// TIA Portal project "Szachy_v2" (V14)

(* hardware
DEVICE "S71500/ET200MP station_1"  S7-1500 station
   slot 0: "Rail_0"  Rack  6ES7 590-1***0-0AA0
   slot 1: "PLC_1"  CPU 1511-1 PN  6ES7 511-1AK00-0AB0  V1.8
      slot 3: "CPU display_1"  6ES7591-1AA00-0AA0
   slot 2: "DI 16x24VDC HF_1"  DI 16x24VDC HF  6ES7 521-1BH00-0AB0  V2.1
   slot 3: "DQ 16x24VDC/0.5A ST_1"  DQ 16x24VDC/0.5A ST  6ES7 522-1BH00-0AB0  V2.0
   slot 4: "AI 4xU/I/RTD/TC ST_1"  AI 4xU/I/RTD/TC ST  6ES7 531-7QD00-0AB0  V1.0
DEVICE "HMI_1"  TP700 Comfort
   slot 0: "TP700 Comfort"  TP700 Comfort  6AV2 124-0GC01-0AX0  14.0.1.0
   slot 1: "HMI_RT_1"  TP700 Comfort  6AV2 124-0GC01-0AX0  14.0.1.0
   slot 5: "HMI_1.IE_CP_1"  PROFINET Interface  14.0.1.0
      slot 1: "PROFINET Interface_1"  PROFINET Interface
         slot 1: "Port_1"  Port
         slot 2: "Port_2"  Port
   slot 7: "HMI_1.MPI/DP_CP_1"  MPI/DP Interface  14.0.1.0
*)

// ===== PLC "PLC_1"  CPU 1511-1 PN =====

VAR_GLOBAL   // PLC tag table "Default tag table"
   "Tag_1" AT %M100.0 : Bool;
   "Tag_2" AT %M100.1 : Bool;
END_VAR

TYPE "Szachownica"
   STRUCT
      figury : Array[0..31] of "Figura";
      pozycja_wybranego_1 : "Pozycja";
      pozycja_wybranego_2 : "Pozycja";
   END_STRUCT;
END_TYPE

TYPE "Figura"
   STRUCT
      kolor : Bool;   // 0-czarny / 1-biały
      rodzaj : Int;   // 0-pawn /1-bishop /2-horse /3-tower / 4-queen /5-king
      zywy : Bool;   // 1-zywy /0-zbity
      mozliwe_ruchy : Array[0..26] of "Pozycja";
      pozycja : "Pozycja";
      poczatkowa_pozycja : Bool := true;
      tura_1_ruchu_piona : Int;
   END_STRUCT;
END_TYPE

TYPE "Pozycja"
   STRUCT
      x : Int;
      y : Int;
   END_STRUCT;
END_TYPE

DATA_BLOCK "StatusyHMI"   // DB1
{ S7_Optimized_Access := 'FALSE' }
VERSION : 0.1
   VAR
      przyciski : Array[0..63] of Bool;
      "statusy figur" : Array[0..63] of Int;
      "przyciski widocznosc" : Array[0..63] of Bool;
   END_VAR
BEGIN
   "przyciski widocznosc"[0] := true;
   "przyciski widocznosc"[1] := true;
   "przyciski widocznosc"[2] := true;
   "przyciski widocznosc"[3] := true;
   "przyciski widocznosc"[4] := true;
   "przyciski widocznosc"[5] := true;
   "przyciski widocznosc"[6] := true;
   "przyciski widocznosc"[7] := true;
   "przyciski widocznosc"[8] := true;
   "przyciski widocznosc"[9] := true;
   "przyciski widocznosc"[10] := true;
   "przyciski widocznosc"[11] := true;
   "przyciski widocznosc"[12] := true;
   "przyciski widocznosc"[13] := true;
   "przyciski widocznosc"[14] := true;
   "przyciski widocznosc"[15] := true;
   "przyciski widocznosc"[16] := true;
   "przyciski widocznosc"[17] := true;
   "przyciski widocznosc"[18] := true;
   "przyciski widocznosc"[19] := true;
   "przyciski widocznosc"[20] := true;
   "przyciski widocznosc"[21] := true;
   "przyciski widocznosc"[22] := true;
   "przyciski widocznosc"[23] := true;
   "przyciski widocznosc"[24] := true;
   "przyciski widocznosc"[25] := true;
   "przyciski widocznosc"[26] := true;
   "przyciski widocznosc"[27] := true;
   "przyciski widocznosc"[28] := true;
   "przyciski widocznosc"[29] := true;
   "przyciski widocznosc"[30] := true;
   "przyciski widocznosc"[31] := true;
   "przyciski widocznosc"[32] := true;
   "przyciski widocznosc"[33] := true;
   "przyciski widocznosc"[34] := true;
   "przyciski widocznosc"[35] := true;
   "przyciski widocznosc"[36] := true;
   "przyciski widocznosc"[37] := true;
   "przyciski widocznosc"[38] := true;
   "przyciski widocznosc"[39] := true;
   "przyciski widocznosc"[40] := true;
   "przyciski widocznosc"[41] := true;
   "przyciski widocznosc"[42] := true;
   "przyciski widocznosc"[43] := true;
   "przyciski widocznosc"[44] := true;
   "przyciski widocznosc"[45] := true;
   "przyciski widocznosc"[46] := true;
   "przyciski widocznosc"[47] := true;
   "przyciski widocznosc"[48] := true;
   "przyciski widocznosc"[49] := true;
   "przyciski widocznosc"[50] := true;
   "przyciski widocznosc"[51] := true;
   "przyciski widocznosc"[52] := true;
   "przyciski widocznosc"[53] := true;
   "przyciski widocznosc"[54] := true;
   "przyciski widocznosc"[55] := true;
   "przyciski widocznosc"[56] := true;
   "przyciski widocznosc"[57] := true;
   "przyciski widocznosc"[58] := true;
   "przyciski widocznosc"[59] := true;
   "przyciski widocznosc"[60] := true;
   "przyciski widocznosc"[61] := true;
   "przyciski widocznosc"[62] := true;
   "przyciski widocznosc"[63] := true;
   "statusy figur"[0] := 12;
   "statusy figur"[1] := 12;
   "statusy figur"[2] := 12;
   "statusy figur"[3] := 12;
   "statusy figur"[4] := 12;
   "statusy figur"[5] := 12;
   "statusy figur"[6] := 12;
   "statusy figur"[7] := 12;
   "statusy figur"[8] := 12;
   "statusy figur"[9] := 12;
   "statusy figur"[10] := 12;
   "statusy figur"[11] := 12;
   "statusy figur"[12] := 12;
   "statusy figur"[13] := 12;
   "statusy figur"[14] := 12;
   "statusy figur"[15] := 12;
   "statusy figur"[16] := 12;
   "statusy figur"[17] := 12;
   "statusy figur"[18] := 12;
   "statusy figur"[19] := 12;
   "statusy figur"[20] := 12;
   "statusy figur"[21] := 12;
   "statusy figur"[22] := 12;
   "statusy figur"[23] := 12;
   "statusy figur"[24] := 12;
   "statusy figur"[25] := 12;
   "statusy figur"[26] := 12;
   "statusy figur"[27] := 12;
   "statusy figur"[28] := 12;
   "statusy figur"[29] := 12;
   "statusy figur"[30] := 12;
   "statusy figur"[31] := 12;
   "statusy figur"[32] := 12;
   "statusy figur"[33] := 12;
   "statusy figur"[34] := 12;
   "statusy figur"[35] := 12;
   "statusy figur"[36] := 12;
   "statusy figur"[37] := 12;
   "statusy figur"[38] := 12;
   "statusy figur"[39] := 12;
   "statusy figur"[40] := 12;
   "statusy figur"[41] := 12;
   "statusy figur"[42] := 12;
   "statusy figur"[43] := 12;
   "statusy figur"[44] := 12;
   "statusy figur"[45] := 12;
   "statusy figur"[46] := 12;
   "statusy figur"[47] := 12;
   "statusy figur"[48] := 12;
   "statusy figur"[49] := 12;
   "statusy figur"[50] := 12;
   "statusy figur"[51] := 12;
   "statusy figur"[52] := 12;
   "statusy figur"[53] := 12;
   "statusy figur"[54] := 12;
   "statusy figur"[55] := 12;
   "statusy figur"[56] := 12;
   "statusy figur"[57] := 12;
   "statusy figur"[58] := 12;
   "statusy figur"[59] := 12;
   "statusy figur"[60] := 12;
   "statusy figur"[61] := 12;
   "statusy figur"[62] := 12;
   "statusy figur"[63] := 12;
END_DATA_BLOCK

DATA_BLOCK "Historia_gry"   // DB3
{ S7_Optimized_Access := 'TRUE' }
VERSION : 0.1
   VAR
      stan_figur : Array[0..200] of "Szachownica";
      indeks_historii : Int := 0;
   END_VAR
BEGIN
END_DATA_BLOCK

DATA_BLOCK "Status_rozgrywki"   // DB4
{ S7_Optimized_Access := 'TRUE' }
VERSION : 0.1
   VAR
      tura_int : Int;
      inicjalizacja : Bool := true;
      Szachownica : "Szachownica";
      tura_bool : Bool := true;   // true - biale false -czarne
      szach_biale : Bool;
      szach_czarne : Bool;
      szachmat_biale : Bool;
      szachmat_czarne : Bool;
      remis : Bool;   // 1- remis, 0 - nie stwierdzono
      status_zakonczenia_gry : Bool;   // 0 - trwa, 1-zakonczono
      komunikat_koniec_gry : Int;   // 0 - wygrana białe, 1- czarne , 2 -remis
      wybrano_pierwszy : Bool;
      indeks1 : Int := -1;
      indeks2 : Int := -2;
      wybrano_drugi : Bool;
   END_VAR
BEGIN
END_DATA_BLOCK

DATA_BLOCK "Inicjalizacja_DB"   // DB5
{ S7_Optimized_Access := 'TRUE' }
VERSION : 0.1
// stored: InstanceOfName Inicjalizacja
"Inicjalizacja"
BEGIN
   Fig_init.figury[7].pozycja.y := 1;
   Fig_init.figury[7].pozycja.x := 8;
   Fig_init.figury[12].pozycja.y := 2;
END_DATA_BLOCK

DATA_BLOCK "sprawdz_czy_remis_DB"   // DB7
{ S7_Optimized_Access := 'TRUE' }
VERSION : 0.1
// stored: InstanceOfName sprawdz_czy_remis
"sprawdz_czy_remis"
BEGIN
END_DATA_BLOCK

// folder: AI

DATA_BLOCK "Ruchy_AI"   // DB8
{ S7_Optimized_Access := 'TRUE' }
VERSION : 0.1
   VAR
      ruchy_1 : Array[0..1] of Bool;
   END_VAR
BEGIN
END_DATA_BLOCK

// folder: (top level)

FUNCTION_BLOCK "Inicjalizacja"   // FB1, SCL
{ S7_Optimized_Access := 'TRUE' }
VERSION : 0.1
   VAR RETAIN
      Fig_init : "Szachownica";
   END_VAR
   VAR
      biale_init : Bool;
   END_VAR
   // Fig_init.figury[0].kolor := 1;
   // Fig_init.figury[0].rodzaj := 3;
   // Fig_init.figury[0].zywy := 1;
   // Fig_init.figury[1].rodzaj := 2;
   // Fig_init.figury[2].rodzaj := 1;
   // Fig_init.figury[3].rodzaj := 4;
   // Fig_init.figury[4].rodzaj := 5;
   // Fig_init.figury[5].rodzaj := 1;
   // Fig_init.figury[6].rodzaj := 2;
   // Fig_init.figury[7].rodzaj := 3;
   // Fig_init.figury[1].zywy := 1;
   // Fig_init.figury[2].zywy := 1;
   // Fig_init.figury[3].zywy := 1;
   // Fig_init.figury[4].zywy := 1;
   // Fig_init.figury[5].zywy := 1;
   // Fig_init.figury[6].zywy := 1;
   // Fig_init.figury[7].zywy := 1;
   // Fig_init.figury[7].kolor := 1;
   // Fig_init.figury[6].kolor := 1;
   // Fig_init.figury[5].kolor := 1;
   // Fig_init.figury[4].kolor := 1;
   // Fig_init.figury[3].kolor := 1;
   // Fig_init.figury[2].kolor := 1;
   // Fig_init.figury[1].kolor := 1;
   // Fig_init.figury[1].pozycja.x := 2;
   // Fig_init.figury[2].pozycja.x := 3;
   // Fig_init.figury[3].pozycja.x := 4;
   // Fig_init.figury[4].pozycja.x := 5;
   // Fig_init.figury[5].pozycja.x := 6;
   // Fig_init.figury[6].pozycja.x := 7;
   // Fig_init.figury[7].pozycja.x := 7;
   // Fig_init.figury[8].pozycja.x := 1;
   // Fig_init.figury[0].pozycja.x := 1;
   // Fig_init.figury[0].pozycja.y := 1;
   // Fig_init.figury[1].pozycja.y := 1;
   // Fig_init.figury[2].pozycja.y := 1;
   // Fig_init.figury[3].pozycja.y := 1;
   // Fig_init.figury[4].pozycja.y := 1;
   // Fig_init.figury[5].pozycja.y := 1;
   // Fig_init.figury[6].pozycja.y := 1;
   // Fig_init.figury[8].kolor := 1;
   // Fig_init.figury[8].zywy := 1;
   // Fig_init.figury[8].pozycja.y := 2;
   // Fig_init.figury[9].kolor := 1;
   // Fig_init.figury[9].rodzaj := 0;
   // Fig_init.figury[9].zywy := 1;
   // Fig_init.figury[10].kolor := 1;
   // Fig_init.figury[10].rodzaj := 0;
   // Fig_init.figury[10].zywy := 1;
   // Fig_init.figury[11].kolor := 1;
   // Fig_init.figury[11].rodzaj := 0;
   // Fig_init.figury[11].zywy := 1;
   // Fig_init.figury[12].kolor := 1;
   // Fig_init.figury[12].rodzaj := 0;
   // Fig_init.figury[12].zywy := 1;
   // Fig_init.figury[13].kolor := 1;
   // Fig_init.figury[13].rodzaj := 0;
   // Fig_init.figury[13].zywy := 1;
   // Fig_init.figury[14].kolor := 1;
   // Fig_init.figury[14].rodzaj := 0;
   // Fig_init.figury[14].zywy := 1;
   // Fig_init.figury[15].kolor := 1;
   // Fig_init.figury[15].rodzaj := 0;
   // Fig_init.figury[15].zywy := 1;
   // Fig_init.figury[9].pozycja.x := 2;
   // Fig_init.figury[9].pozycja.y := 2;
   // Fig_init.figury[10].pozycja.x := 3;
   // Fig_init.figury[10].pozycja.y := 2;
   // Fig_init.figury[11].pozycja.x := 4;
   // Fig_init.figury[11].pozycja.y := 2;
   // Fig_init.figury[12].pozycja.x := 5;
   // Fig_init.figury[13].pozycja.x := 6;
   // Fig_init.figury[13].pozycja.y := 2;
   // Fig_init.figury[14].pozycja.x := 7;
   // Fig_init.figury[14].pozycja.y := 2;
   // Fig_init.figury[15].pozycja.x := 8;
   // Fig_init.figury[15].pozycja.y := 2;
   // Fig_init.figury[16].kolor := 0;
   // Fig_init.figury[16].zywy := 1;
   // Fig_init.figury[17].kolor := 0;
   // Fig_init.figury[17].rodzaj := 0;
   // Fig_init.figury[17].zywy := 1;
   // Fig_init.figury[23].kolor := 0;
   // Fig_init.figury[23].rodzaj := 0;
   // Fig_init.figury[23].zywy := 1;
   // Fig_init.figury[18].kolor := 0;
   // Fig_init.figury[18].rodzaj := 0;
   // Fig_init.figury[18].zywy := 1;
   // Fig_init.figury[19].kolor := 0;
   // Fig_init.figury[19].rodzaj := 0;
   // Fig_init.figury[19].zywy := 1;
   // Fig_init.figury[22].kolor := 0;
   // Fig_init.figury[22].rodzaj := 0;
   // Fig_init.figury[22].zywy := 1;
   // Fig_init.figury[21].kolor := 0;
   // Fig_init.figury[21].rodzaj := 0;
   // Fig_init.figury[21].zywy := 1;
   // Fig_init.figury[20].kolor := 0;
   // Fig_init.figury[20].rodzaj := 0;
   // Fig_init.figury[20].zywy := 1;
   // Fig_init.figury[16].pozycja.x := 1;
   // Fig_init.figury[16].pozycja.y := 7;
   // Fig_init.figury[17].pozycja.x := 2;
   // Fig_init.figury[17].pozycja.y := 7;
   // Fig_init.figury[18].pozycja.x := 3;
   // Fig_init.figury[18].pozycja.y := 7;
   // Fig_init.figury[19].pozycja.x := 4;
   // Fig_init.figury[19].pozycja.y := 7;
   // Fig_init.figury[20].pozycja.x := 5;
   // Fig_init.figury[20].pozycja.y := 7;
   // Fig_init.figury[21].pozycja.x := 6;
   // Fig_init.figury[21].pozycja.y := 7;
   // Fig_init.figury[22].pozycja.x := 7;
   // Fig_init.figury[22].pozycja.y := 7;
   // Fig_init.figury[23].pozycja.x := 8;
   // Fig_init.figury[23].pozycja.y := 7;
   // Fig_init.figury[24].kolor := 0;
   // Fig_init.figury[24].zywy := 1;
   // Fig_init.figury[24].rodzaj := 3;
   // Fig_init.figury[25].kolor := 0;
   // Fig_init.figury[25].rodzaj := 2;
   // Fig_init.figury[25].zywy := 1;
   // Fig_init.figury[24].pozycja.x := 1;
   // Fig_init.figury[24].pozycja.y := 8;
   // Fig_init.figury[25].pozycja.x := 2;
   // Fig_init.figury[25].pozycja.y := 8;
   // Fig_init.figury[26].kolor := 0;
   // Fig_init.figury[26].rodzaj := 1;
   // Fig_init.figury[26].zywy := 1;
   // Fig_init.figury[26].pozycja.x := 3;
   // Fig_init.figury[26].pozycja.y := 8;
   // Fig_init.figury[27].kolor := 0;
   // Fig_init.figury[27].rodzaj := 4;
   // Fig_init.figury[27].zywy := 1;
   // Fig_init.figury[27].pozycja.x := 4;
   // Fig_init.figury[27].pozycja.y := 8;
   // Fig_init.figury[28].kolor := 0;
   // Fig_init.figury[28].rodzaj := 5;
   // Fig_init.figury[28].zywy := 1;
   // Fig_init.figury[28].pozycja.x := 5;
   // Fig_init.figury[28].pozycja.y := 8;
   // Fig_init.figury[29].kolor := 0;
   // Fig_init.figury[29].rodzaj := 1;
   // Fig_init.figury[29].zywy := 1;
   // Fig_init.figury[29].pozycja.x := 6;
   // Fig_init.figury[29].pozycja.y := 8;
   // Fig_init.figury[30].kolor := 0;
   // Fig_init.figury[30].rodzaj := 2;
   // Fig_init.figury[30].zywy := 1;
   // Fig_init.figury[30].pozycja.x := 7;
   // Fig_init.figury[30].pozycja.y := 8;
   // Fig_init.figury[31].kolor := 0;
   // Fig_init.figury[31].rodzaj := 3;
   // Fig_init.figury[31].zywy := 1;
   // Fig_init.figury[31].pozycja.x := 8;
   // Fig_init.figury[31].pozycja.y := 8;
BEGIN
   "Historia_gry".stan_figur[0] := #Fig_init;
   "Status_rozgrywki".Szachownica := #Fig_init;
   "Status_rozgrywki".tura_int := 1;
   "Status_rozgrywki".inicjalizacja := false;
   "Status_rozgrywki".tura_bool := TRUE;
   "Czyszczenie_mozliwych_ruchów"();
   "Czyszczenie_podświetlenia"();
   #biale_init := TRUE;
   "Status_rozgrywki".szach_biale := 0;
   "Status_rozgrywki".szach_czarne := 0;
   "Status_rozgrywki".szachmat_biale := 0;
   "Status_rozgrywki".szachmat_czarne := 0;
   "Status_rozgrywki".status_zakonczenia_gry := 0;
   "Status_rozgrywki".komunikat_koniec_gry := 0;
END_FUNCTION_BLOCK

FUNCTION "tura_biale" : Void   // FC1, SCL
{ S7_Optimized_Access := 'TRUE' }
VERSION : 0.1
   VAR_IN_OUT
      tura : Bool;
   END_VAR
   VAR_TEMP
      ilosc_mozliwych_ruchow : Int;
      figura_ruch : "Figura";
      tura_zbocze : Bool;
   END_VAR
BEGIN
   "tura_biale_trig_DB"(CLK := #tura,
                         Q => #tura_zbocze);
   //"Status_rozgrywki".szach_biale := "sprawdz_czy_szach"(tura_bool := TRUE, szachownica := "Status_rozgrywki".Szachownica);
   //#ilosc_mozliwych_ruchow := "Wykrywanie_ruchów"(tura_bool := TRUE, Szachownica := "Status_rozgrywki".Szachownica);
   //"Status_rozgrywki".szachmat_biale := (#ilosc_mozliwych_ruchow = 0);

    IF #tura_zbocze OR "Inicjalizacja_DB".biale_init THEN
           "Status_rozgrywki".szach_biale := "sprawdz_czy_szach"(tura_bool := TRUE, szachownica := "Status_rozgrywki".Szachownica);
           #ilosc_mozliwych_ruchow := "Wykrywanie_ruchów"(tura_bool := TRUE, Szachownica := "Status_rozgrywki".Szachownica);
           "Status_rozgrywki".szachmat_biale := (#ilosc_mozliwych_ruchow = 0 AND "Status_rozgrywki".szach_biale);

           "Inicjalizacja_DB".biale_init := FALSE;
       END_IF;
    IF #tura THEN
       IF "Status_rozgrywki".wybrano_pierwszy AND "Status_rozgrywki".wybrano_drugi THEN
           IF "konwersja_pozycja_na_figura"(pozycja := "Status_rozgrywki".Szachownica.pozycja_wybranego_1,
                                                Szachownica := "Status_rozgrywki".Szachownica, figura => #figura_ruch) THEN
               IF "sprawdz_czy_ruch_mozliwy"(Szachownica := "Status_rozgrywki".Szachownica, figura := #figura_ruch, pozycja := "Status_rozgrywki".Szachownica.pozycja_wybranego_2) THEN
                   "wykonanie_ruchu"(pozycja := "Status_rozgrywki".Szachownica.pozycja_wybranego_2,
                                     szachownica := "Status_rozgrywki".Szachownica,
                                     figura := #figura_ruch);
                   "Czyszczenie_podświetlenia"();
                   "Czyszczenie_mozliwych_ruchów"();
                   "Status_rozgrywki".tura_int += 1;
                   "Status_rozgrywki".szach_biale := 0;
                   #tura := false;
               END_IF;
           END_IF;
       END_IF;
   END_IF;
END_FUNCTION

FUNCTION "tura_czarne" : Void   // FC2, SCL
{ S7_Optimized_Access := 'TRUE' }
VERSION : 0.1
   VAR_IN_OUT
      tura : Bool;
   END_VAR
   VAR_TEMP
      ilosc_mozliwych_ruchow : Int;
      figura_ruch : "Figura";
      tura_zbocze : Bool;
   END_VAR
BEGIN
   "Tura_czarne_trug_DB"(CLK:=#tura,
                         Q=>#tura_zbocze);
   //"Status_rozgrywki".szach_czarne := "sprawdz_czy_szach"(tura_bool := FALSE, szachownica := "Status_rozgrywki".Szachownica);
   //#ilosc_mozliwych_ruchow := "Wykrywanie_ruchów"(tura_bool := FALSE, Szachownica := "Status_rozgrywki".Szachownica);
   //"Status_rozgrywki".szachmat_czarne := (#ilosc_mozliwych_ruchow = 0);
   IF #tura_zbocze THEN
       "Status_rozgrywki".szach_czarne := "sprawdz_czy_szach"(tura_bool := FALSE, szachownica := "Status_rozgrywki".Szachownica);
       #ilosc_mozliwych_ruchow := "Wykrywanie_ruchów"(tura_bool := FALSE, Szachownica := "Status_rozgrywki".Szachownica);
       "Status_rozgrywki".szachmat_czarne := (#ilosc_mozliwych_ruchow = 0 AND "Status_rozgrywki".szach_czarne);
       "sprawdz_czy_remis_DB"(#ilosc_mozliwych_ruchow);
   END_IF;
   IF NOT #tura THEN
       IF "Status_rozgrywki".wybrano_pierwszy AND "Status_rozgrywki".wybrano_drugi THEN
           IF "konwersja_pozycja_na_figura"(pozycja := "Status_rozgrywki".Szachownica.pozycja_wybranego_1,
                                                Szachownica := "Status_rozgrywki".Szachownica, figura => #figura_ruch) THEN
               IF "sprawdz_czy_ruch_mozliwy"(Szachownica := "Status_rozgrywki".Szachownica, figura := #figura_ruch, pozycja := "Status_rozgrywki".Szachownica.pozycja_wybranego_2) THEN
                   "wykonanie_ruchu"(pozycja := "Status_rozgrywki".Szachownica.pozycja_wybranego_2,
                                     szachownica := "Status_rozgrywki".Szachownica,
                                     figura := #figura_ruch);
                   "Czyszczenie_podświetlenia"();
                   "Czyszczenie_mozliwych_ruchów"();
                   "Status_rozgrywki".tura_int += 1;
                   "Status_rozgrywki".szach_czarne := 0;
                   #tura := true;
               END_IF;
           END_IF;
       END_IF;
   END_IF;
END_FUNCTION

FUNCTION "ObslugaHMI" : Void   // FC24, SCL
{ S7_Optimized_Access := 'TRUE' }
VERSION : 0.1
BEGIN
   "Czytanie_wcisnietych_przyciskow"();
   "Statusy figur"("Status_rozgrywki".Szachownica);
   "Ukrywanie_przycisków"("Status_rozgrywki".Szachownica);

   IF "Status_rozgrywki".szachmat_biale THEN
       "Status_rozgrywki".komunikat_koniec_gry := 0;
       "Status_rozgrywki".status_zakonczenia_gry := 1;
   ELSIF "Status_rozgrywki".szachmat_czarne THEN
       "Status_rozgrywki".komunikat_koniec_gry := 1;
       "Status_rozgrywki".status_zakonczenia_gry := 1;
   ELSIF "Status_rozgrywki".remis THEN
       "Status_rozgrywki".komunikat_koniec_gry := 2;
       "Status_rozgrywki".status_zakonczenia_gry := 1;
   END_IF;
END_FUNCTION

ORGANIZATION_BLOCK "Main"   // OB1, LAD, ProgramCycle
TITLE = "Main Program Sweep (Cycle)"
{ S7_Optimized_Access := 'TRUE' }
VERSION : 0.1
   VAR_INPUT
      Initial_Call : Bool;   // Initial call of this OB
      Remanence : Bool;   // =True, if remanent data are available
   END_VAR
BEGIN

REGION Network 1: Inicjalizacja pozycji figur
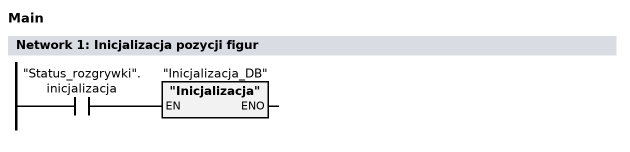
   RUNG wire#powerrail
      Contact( "Status_rozgrywki".inicjalizacja )
      "Inicjalizacja_DB"()
   END_RUNG
   // the same network as SCL:
   IF "Status_rozgrywki".inicjalizacja THEN
       "Inicjalizacja_DB"();   // "Inicjalizacja"
   END_IF;
END_REGION
END_ORGANIZATION_BLOCK

ORGANIZATION_BLOCK "Cyclic interrupt"   // OB30, LAD, CyclicInterrupt
{ S7_Optimized_Access := 'TRUE' }
VERSION : 0.1
   VAR_INPUT
      Initial_Call : Bool;   // Initial call of this OB
      Event_Count : Int;   // Events discarded
   END_VAR
BEGIN

REGION Network 1
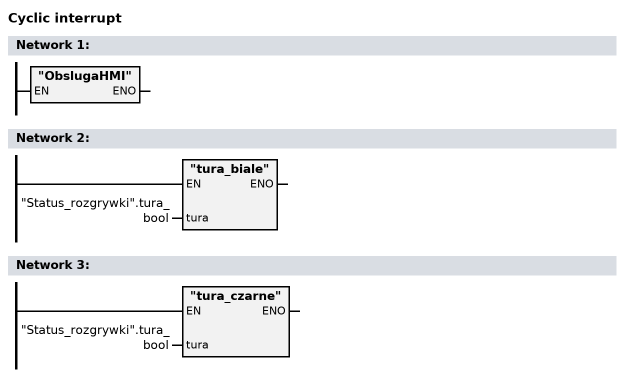
   RUNG wire#powerrail
      "ObslugaHMI"()
   END_RUNG
   // the same network as SCL:
   "ObslugaHMI"();
END_REGION

REGION Network 2
   RUNG wire#powerrail
      "tura_biale"(tura := "Status_rozgrywki".tura_bool)
   END_RUNG
   // the same network as SCL:
   "tura_biale"(tura := "Status_rozgrywki".tura_bool);
END_REGION

REGION Network 3
   RUNG wire#powerrail
      "tura_czarne"(tura := "Status_rozgrywki".tura_bool)
   END_RUNG
   // the same network as SCL:
   "tura_czarne"(tura := "Status_rozgrywki".tura_bool);
END_REGION
END_ORGANIZATION_BLOCK

// folder: AI

FUNCTION "przepisanie_ruchów_do_tabeli" : Void   // FC34, SCL
{ S7_Optimized_Access := 'TRUE' }
VERSION : 0.1
BEGIN
END_FUNCTION

// folder: Obsluga Hmi

FUNCTION "Czytanie_wcisnietych_przyciskow" : Void   // FC4, SCL
{ S7_Optimized_Access := 'TRUE' }
VERSION : 0.1
   VAR_TEMP
      i : Int;
      wybrano_pierwszy : Bool;
      wybrano_drugi : Bool;
   END_VAR
BEGIN

   FOR #i := 0 TO 63 DO
       IF "StatusyHMI".przyciski[#i] AND NOT "Status_rozgrywki".wybrano_pierwszy THEN
           "Status_rozgrywki".indeks1 := #i;
           "Status_rozgrywki".wybrano_pierwszy := true;
           "Status_rozgrywki".Szachownica.pozycja_wybranego_1 := "konwersja_indeks_na_xy"(#i);

       END_IF;
       IF "StatusyHMI".przyciski[#i] AND "Status_rozgrywki".wybrano_pierwszy
           AND NOT ("Status_rozgrywki".indeks1 = #i) THEN
           "Status_rozgrywki".indeks2 := #i;
           "Status_rozgrywki".wybrano_drugi := true;
           "Status_rozgrywki".Szachownica.pozycja_wybranego_2 := "konwersja_indeks_na_xy"(#i);
       END_IF;
   END_FOR;
   IF NOT ("Status_rozgrywki".indeks1 = -1) THEN
       IF "StatusyHMI".przyciski["Status_rozgrywki".indeks1] = false THEN
           IF "Status_rozgrywki".wybrano_drugi THEN
               "Status_rozgrywki".Szachownica.pozycja_wybranego_2.x := 0;
               "Status_rozgrywki".Szachownica.pozycja_wybranego_2.y := 0;
               "Status_rozgrywki".indeks2 := -2;
               "Status_rozgrywki".wybrano_drugi := FALSE;
           END_IF;
           "Status_rozgrywki".wybrano_pierwszy := FALSE;
           "Status_rozgrywki".Szachownica.pozycja_wybranego_1.x := 0;
           "Status_rozgrywki".Szachownica.pozycja_wybranego_1.y := 0;
           "Status_rozgrywki".indeks1 := -1;

       END_IF;
   END_IF;
   IF NOT ("Status_rozgrywki".indeks2 = -2) THEN
       IF "StatusyHMI".przyciski["Status_rozgrywki".indeks2] = false THEN
           "Status_rozgrywki".indeks2 := -2;
           "Status_rozgrywki".wybrano_drugi := FALSE;
           "Status_rozgrywki".Szachownica.pozycja_wybranego_2.x :=
           "Status_rozgrywki".Szachownica.pozycja_wybranego_2.y := 0;
       END_IF;
   END_IF;
END_FUNCTION

FUNCTION "Statusy figur" : Void   // FC25, SCL
{ S7_Optimized_Access := 'TRUE' }
VERSION : 0.1
   VAR_INPUT
      Szachownica : "Szachownica";
   END_VAR
   VAR_TEMP
      i : Int;
      indeks : Int;
   END_VAR
BEGIN
   FOR #i := 0 TO 63 DO
       "StatusyHMI"."statusy figur"[#i] := 12 ;
   END_FOR;
   FOR #i := 0 TO 31 DO
       IF #Szachownica.figury[#i].zywy = true THEN
           #indeks := 63 - (#Szachownica.figury[#i].pozycja.y * 8) + #Szachownica.figury[#i].pozycja.x;
           IF #Szachownica.figury[#i].kolor = 1 THEN
               "StatusyHMI"."statusy figur"[#indeks] := #Szachownica.figury[#i].rodzaj;
           ELSE
               "StatusyHMI"."statusy figur"[#indeks] := #Szachownica.figury[#i].rodzaj + 6 ;
           END_IF;
    //   ELSE
     //      "StatusyHMI"."statusy figur"[#i] := 12;
       END_IF;
   END_FOR;
END_FUNCTION

FUNCTION "podświetlenie pól" : Void   // FC26, SCL
{ S7_Optimized_Access := 'TRUE' }
VERSION : 0.1
BEGIN
END_FUNCTION

FUNCTION "konwersja_indeks_na_xy" : "Pozycja"   // FC29, SCL
{ S7_Optimized_Access := 'TRUE' }
VERSION : 0.1
   VAR_INPUT
      indeks : Int;
   END_VAR
   VAR_TEMP
      i : Int;
   END_VAR
BEGIN
   #konwersja_indeks_na_xy.x := 0;
   #konwersja_indeks_na_xy.y := 0;

   WHILE #konwersja_indeks_na_xy.y *8 <= #indeks DO
       #konwersja_indeks_na_xy.y += 1;
   END_WHILE;
   #konwersja_indeks_na_xy.x := #indeks +1 - 8*(#konwersja_indeks_na_xy.y-1);
END_FUNCTION

FUNCTION "Ukrywanie_przycisków" : Void   // FC33, SCL
{ S7_Optimized_Access := 'TRUE' }
VERSION : 0.1
   VAR_INPUT
      Szachownica : "Szachownica";
   END_VAR
   VAR_TEMP
      i : Int;
      indeks : Int;
   END_VAR
BEGIN

   REGION biale_1_ruch
       IF "Status_rozgrywki".tura_bool AND NOT "Status_rozgrywki".wybrano_pierwszy THEN
           FOR #i := 0 TO 63 DO
               "StatusyHMI"."przyciski widocznosc"[#i] := false;
           END_FOR;
           FOR #i := 0 TO 15 DO
               IF #Szachownica.figury[#i].zywy = true THEN
                   #indeks := 63 - (#Szachownica.figury[#i].pozycja.y * 8) + #Szachownica.figury[#i].pozycja.x;
                   IF #Szachownica.figury[#i].kolor = 1 THEN
                       "StatusyHMI"."przyciski widocznosc"[#indeks] := true;
                   END_IF;
               END_IF;
           END_FOR;
       END_IF;
   END_REGION ;
   REGION biale_2_ruch
       IF "Status_rozgrywki".tura_bool AND "Status_rozgrywki".wybrano_pierwszy THEN
           FOR #i := 0 TO 63 DO
               "StatusyHMI"."przyciski widocznosc"[#i] := TRUE;
           END_FOR;
           FOR #i := 0 TO 15 DO
               IF #Szachownica.figury[#i].zywy = true THEN
                   #indeks := 63 - (#Szachownica.figury[#i].pozycja.y * 8) + #Szachownica.figury[#i].pozycja.x;
                   IF #Szachownica.figury[#i].kolor = 1  AND NOT ("Status_rozgrywki".Szachownica.pozycja_wybranego_1.x =
                       #Szachownica.figury[#i].pozycja.x AND "Status_rozgrywki".Szachownica.pozycja_wybranego_1.y =
                       #Szachownica.figury[#i].pozycja.y) THEN
                       "StatusyHMI"."przyciski widocznosc"[#indeks] := false;
                   END_IF;
               END_IF;
           END_FOR;
       END_IF;
   END_REGION ;
   REGION czarne_1_ruch
       IF NOT "Status_rozgrywki".tura_bool AND NOT "Status_rozgrywki".wybrano_pierwszy THEN
           FOR #i := 0 TO 63 DO
               "StatusyHMI"."przyciski widocznosc"[#i] := false;
           END_FOR;
           FOR #i := 16 TO 31 DO
               IF #Szachownica.figury[#i].zywy = true THEN
                   #indeks := 63 - (#Szachownica.figury[#i].pozycja.y * 8) + #Szachownica.figury[#i].pozycja.x;
                   IF #Szachownica.figury[#i].kolor = false THEN
                       "StatusyHMI"."przyciski widocznosc"[#indeks] := true;
                   END_IF;
               END_IF;
           END_FOR;
       END_IF;
   END_REGION ;
   REGION czarne_2_ruch
       IF NOT "Status_rozgrywki".tura_bool AND "Status_rozgrywki".wybrano_pierwszy THEN
           FOR #i := 0 TO 63 DO
               "StatusyHMI"."przyciski widocznosc"[#i] := TRUE;
           END_FOR;
           FOR #i := 16 TO 31 DO
               IF #Szachownica.figury[#i].zywy = true THEN
                   #indeks := 63 - (#Szachownica.figury[#i].pozycja.y* 8) + #Szachownica.figury[#i].pozycja.x;
                   IF #Szachownica.figury[#i].kolor = false AND NOT ("Status_rozgrywki".Szachownica.pozycja_wybranego_1.x =
                       #Szachownica.figury[#i].pozycja.x AND "Status_rozgrywki".Szachownica.pozycja_wybranego_1.y =
                       #Szachownica.figury[#i].pozycja.y) THEN
                       "StatusyHMI"."przyciski widocznosc"[#indeks] := false;
                   END_IF;
               END_IF;
           END_FOR;
       END_IF;
   END_REGION ;
END_FUNCTION

// folder: remis

FUNCTION_BLOCK "sprawdz_czy_remis"   // FB2, SCL
{ S7_Optimized_Access := 'TRUE' }
VERSION : 0.1
   VAR_INPUT
      ilosc_ruchów : Int;
   END_VAR
   VAR
      stwierdzono_remis : Bool := 0;
   END_VAR
BEGIN
   IF #ilosc_ruchów = 0 AND ( (NOT "Status_rozgrywki".szach_biale AND "Status_rozgrywki".tura_bool) OR
       (NOT "Status_rozgrywki".szach_czarne AND NOT "Status_rozgrywki".tura_bool) ) THEN
       #stwierdzono_remis := true;
   END_IF;




   "Status_rozgrywki".remis := #stwierdzono_remis;
END_FUNCTION_BLOCK

// folder: ruch

FUNCTION "wykonanie_ruchu" : Void   // FC27, SCL
{ S7_Optimized_Access := 'TRUE' }
VERSION : 0.1
   VAR_INPUT
      pozycja : "Pozycja";
   END_VAR
   VAR_IN_OUT
      szachownica : "Szachownica";
      figura : "Figura";
   END_VAR
   VAR_TEMP
      i : Int;
   END_VAR
BEGIN
       FOR #i := 0 TO 31 DO
           IF #szachownica.figury[#i].zywy = 1 THEN
               IF #szachownica.figury[#i].pozycja.x = #pozycja.x AND
                   #szachownica.figury[#i].pozycja.y = #pozycja.y THEN
                   #szachownica.figury[#i].zywy := false;
                   #szachownica.figury[#i].pozycja.x := #szachownica.figury[#i].pozycja.y := 0;
                   #szachownica.figury[#i].poczatkowa_pozycja := false;
               END_IF;
               IF #szachownica.figury[#i].pozycja.x = #figura.pozycja.x AND
                   #szachownica.figury[#i].pozycja.y = #figura.pozycja.y THEN
                   #szachownica.figury[#i].pozycja.x := #pozycja.x;
                   #szachownica.figury[#i].pozycja.y := #pozycja.y;
                   #szachownica.figury[#i].poczatkowa_pozycja := false;
               END_IF;
           END_IF;
       END_FOR;
END_FUNCTION

FUNCTION "sprawdz_czy_ruch_mozliwy" : Bool   // FC28, SCL
{ S7_Optimized_Access := 'TRUE' }
VERSION : 0.1
   VAR_INPUT
      pozycja : "Pozycja";
   END_VAR
   VAR_IN_OUT
      figura : "Figura";
      Szachownica : "Szachownica";
   END_VAR
   VAR_TEMP
      i : Int;
      j : Int;
   END_VAR
BEGIN
   #sprawdz_czy_ruch_mozliwy := false;
   REGION Roszada
       IF #figura.rodzaj = 5 THEN
           IF #figura.poczatkowa_pozycja = true THEN
               IF #figura.kolor = true THEN
                   IF #pozycja.x = 3 AND #pozycja.y = 1 THEN
                       FOR #i := 0 TO 26 DO
                           IF #figura.mozliwe_ruchy[#i].x = 3 AND
                               #figura.mozliwe_ruchy[#i].y = 1 THEN
                               #Szachownica.figury[0].pozycja.x := 4;
                               #Szachownica.figury[0].poczatkowa_pozycja := false;
                               #sprawdz_czy_ruch_mozliwy := TRUE;
                           END_IF;
                       END_FOR;
                   ELSIF #pozycja.x = 7 AND #pozycja.y = 1 THEN
                       FOR #i := 0 TO 26 DO
                           IF #figura.mozliwe_ruchy[#i].x = 7 AND
                               #figura.mozliwe_ruchy[#i].y = 1 THEN
                               #Szachownica.figury[7].pozycja.x := 6;
                               #Szachownica.figury[7].poczatkowa_pozycja := false;
                               #sprawdz_czy_ruch_mozliwy := TRUE;
                           END_IF;
                       END_FOR;
                   END_IF;
               ELSE
                   IF #pozycja.x = 3 AND #pozycja.y = 8 THEN
                       FOR #i := 0 TO 26 DO
                           IF #figura.mozliwe_ruchy[#i].x = 3 AND
                               #figura.mozliwe_ruchy[#i].y = 8 THEN
                               #Szachownica.figury[24].pozycja.x := 4;
                               #Szachownica.figury[24].poczatkowa_pozycja := false;
                               #sprawdz_czy_ruch_mozliwy := TRUE;
                           END_IF;
                       END_FOR;
                   ELSIF #pozycja.x = 7 AND #pozycja.y = 8 THEN
                       FOR #i := 0 TO 26 DO
                           IF #figura.mozliwe_ruchy[#i].x = 7 AND
                               #figura.mozliwe_ruchy[#i].y = 8 THEN
                               #Szachownica.figury[31].pozycja.x := 6;
                               #Szachownica.figury[31].poczatkowa_pozycja := false;
                               #sprawdz_czy_ruch_mozliwy := TRUE;
                           END_IF;
                       END_FOR;
                   END_IF;
               END_IF;
           END_IF;
       END_IF;
   END_REGION ;
   REGION Bicie w przelocie 
       IF #figura.rodzaj = 0 THEN
           IF #figura.kolor = true THEN
               IF #pozycja.x = #figura.pozycja.x AND #pozycja.y = #figura.pozycja.y + 2 THEN
                   FOR #i := 0 TO 26 DO
                       IF #figura.mozliwe_ruchy[#i].x = #pozycja.x AND
                           #figura.mozliwe_ruchy[#i].y = #pozycja.y THEN
                           FOR #j := 0 TO 31 DO
                               IF #figura.pozycja.x = #Szachownica.figury[#j].pozycja.x AND
                                   #figura.pozycja.y = #Szachownica.figury[#j].pozycja.y THEN
                                   #Szachownica.figury[#j].tura_1_ruchu_piona := "Status_rozgrywki".tura_int;
                               END_IF;
                           END_FOR;
                       END_IF;
                   END_FOR;
               END_IF;
               FOR #j := 0 TO 31 DO
                   IF #Szachownica.figury[#j].kolor = false THEN
                       IF (#figura.pozycja.x + 1 = #Szachownica.figury[#j].pozycja.x OR
                           #figura.pozycja.x - 1 = #Szachownica.figury[#j].pozycja.x) AND
                           #figura.pozycja.y = #Szachownica.figury[#j].pozycja.y THEN
                           IF #Szachownica.figury[#j].rodzaj = 0 THEN
                               IF #Szachownica.figury[#j].tura_1_ruchu_piona = "Status_rozgrywki".tura_int - 1 THEN
                                   #Szachownica.figury[#j].zywy := false;
                                   #Szachownica.figury[#j].pozycja.x := #Szachownica.figury[#j].pozycja.y := 0;
                                   #sprawdz_czy_ruch_mozliwy := TRUE;
                               END_IF;
                           END_IF;
                       END_IF;
                   END_IF;
               END_FOR;
           ELSE
               IF #pozycja.x = #figura.pozycja.x AND #pozycja.y = #figura.pozycja.y - 2 THEN
                   FOR #i := 0 TO 26 DO
                       IF #figura.mozliwe_ruchy[#i].x = #pozycja.x AND
                           #figura.mozliwe_ruchy[#i].y = #pozycja.y THEN
                           FOR #j := 0 TO 31 DO
                               IF #figura.pozycja.x = #Szachownica.figury[#j].pozycja.x AND
                                   #figura.pozycja.y = #Szachownica.figury[#j].pozycja.y THEN
                                   #Szachownica.figury[#j].tura_1_ruchu_piona := "Status_rozgrywki".tura_int;
                                   #sprawdz_czy_ruch_mozliwy := TRUE;
                               END_IF;
                           END_FOR;
                       END_IF;
                   END_FOR;
               END_IF;
               FOR #j := 0 TO 31 DO
                   IF #Szachownica.figury[#j].kolor = true THEN
                       IF (#figura.pozycja.x + 1 = #Szachownica.figury[#j].pozycja.x OR
                           #figura.pozycja.x - 1 = #Szachownica.figury[#j].pozycja.x) AND
                           #figura.pozycja.y = #Szachownica.figury[#j].pozycja.y THEN
                           IF #Szachownica.figury[#j].rodzaj = 0 THEN
                               IF #Szachownica.figury[#j].tura_1_ruchu_piona = "Status_rozgrywki".tura_int - 1 THEN
                                   #Szachownica.figury[#j].zywy := false;
                                   #Szachownica.figury[#j].pozycja.x := #Szachownica.figury[#j].pozycja.y := 0;
                                   #sprawdz_czy_ruch_mozliwy := TRUE;
                               END_IF;
                           END_IF;
                       END_IF;
                   END_IF;
               END_FOR;
           END_IF;
       END_IF;
   END_REGION;
   FOR #i := 0 TO 26 DO
       IF #figura.mozliwe_ruchy[#i].x = #pozycja.x AND
           #figura.mozliwe_ruchy[#i].y = #pozycja.y THEN
           #sprawdz_czy_ruch_mozliwy := TRUE;
           EXIT;
       END_IF;
   END_FOR;
END_FUNCTION

FUNCTION "konwersja_pozycja_na_figura" : Bool   // FC30, LAD
{ S7_Optimized_Access := 'TRUE' }
VERSION : 0.1
   VAR_INPUT
      pozycja : "Pozycja";
      Szachownica : "Szachownica";
   END_VAR
   VAR_OUTPUT
      figura : "Figura";
   END_VAR
   VAR_TEMP
      i : Int;
   END_VAR
BEGIN

REGION Network 1 (SCL)

   FOR #i := 0 TO 31 DO
       IF #pozycja.x = #Szachownica.figury[#i].pozycja.x AND
           #pozycja.y = #Szachownica.figury[#i].pozycja.y THEN 
           #figura := #Szachownica.figury[#i];
           #konwersja_pozycja_na_figura := true;
           END_IF;
       END_FOR;
END_REGION
END_FUNCTION

FUNCTION "Czyszczenie_podświetlenia" : Void   // FC31, SCL
{ S7_Optimized_Access := 'TRUE' }
VERSION : 0.1
BEGIN
   "StatusyHMI".<??.?> := 0;
   "StatusyHMI".<??.?> := 0;
   "StatusyHMI".<??.?> := 0;
   "StatusyHMI".<??.?> := 0;
   "Status_rozgrywki".Szachownica.pozycja_wybranego_1.x :=
   "Status_rozgrywki".Szachownica.pozycja_wybranego_1.y :=
   "Status_rozgrywki".Szachownica.pozycja_wybranego_2.x :=
   "Status_rozgrywki".Szachownica.pozycja_wybranego_2.y := 0;
   "Status_rozgrywki".indeks1 := -1;
   "Status_rozgrywki".indeks2 := -2;
   "Status_rozgrywki".wybrano_pierwszy := false;
   "Status_rozgrywki".wybrano_drugi := false;
END_FUNCTION

FUNCTION "Czyszczenie_mozliwych_ruchów" : Void   // FC32, SCL
{ S7_Optimized_Access := 'TRUE' }
VERSION : 0.1
   VAR_TEMP
      i : Int;
      j : Int;
      pozycja0 : "Pozycja";
   END_VAR
BEGIN
   #pozycja0.x := #pozycja0.y := 0;
   FOR #i := 0 TO 31 DO
       FOR #j := 0 TO 26 DO
           "Status_rozgrywki".Szachownica.figury[#i].mozliwe_ruchy[#j]:= #pozycja0;
       END_FOR;
   END_FOR;
END_FUNCTION

// folder: wykrywanie_szach

FUNCTION "sprawdz_czy_szach" : Bool   // FC17, SCL
{ S7_Optimized_Access := 'TRUE' }
VERSION : 0.1
   VAR_INPUT
      tura_bool : Bool;
   END_VAR
   VAR_IN_OUT
      szachownica : "Szachownica";
   END_VAR
   VAR_TEMP
      i : Int;
      szach_bialy : Bool;
      szach_czarny : Bool;
   END_VAR
BEGIN
   #szach_bialy := #szach_czarny := false;
   IF NOT #tura_bool THEN
       FOR #i := 0 TO 15 DO
           IF #szachownica.figury[#i].zywy = 1 THEN
               #szach_czarny := "Sprawdz_ruchy_figury_bez_sprawdzania"(szachownica := #szachownica,
                                                                       figura := #szachownica.figury[#i]);
               IF #szach_czarny THEN
                   EXIT;
               END_IF;
           END_IF;
       END_FOR;
   ELSE
       FOR #i := 16 TO 31 DO
           IF "Status_rozgrywki".Szachownica.figury[#i].zywy = 1 THEN
               #szach_bialy := "Sprawdz_ruchy_figury_bez_sprawdzania"(szachownica := #szachownica,
                                                                      figura := #szachownica.figury[#i]);
               IF #szach_bialy THEN
                   EXIT;
               END_IF;
           END_IF;
       END_FOR;
   END_IF;

   #sprawdz_czy_szach := (#szach_bialy OR #szach_czarny);
END_FUNCTION

FUNCTION "sprawdz_czy_pion_szach" : Bool   // FC18, SCL
{ S7_Optimized_Access := 'TRUE' }
VERSION : 0.1
   VAR_INPUT
      szachownica : "Szachownica";
      polozenie_krola : "Pozycja";
   END_VAR
   VAR_IN_OUT
      pion : "Figura";
   END_VAR
   VAR_TEMP
      poz_temp : "Pozycja";
      indeks_mozliwych_ruchow : Int;
   END_VAR
BEGIN
   #indeks_mozliwych_ruchow := 0;
   #sprawdz_czy_pion_szach := false;
   IF #pion.kolor = 1 THEN
       IF #pion.pozycja.y = 2 THEN
           #poz_temp.x := #pion.pozycja.x;
           #poz_temp.y := #pion.pozycja.y + 2;
           IF "sprawdz_czy_na_szachownicy"(#poz_temp) THEN
               IF "sprawdz_czy_wolne"(pozycja := #poz_temp, szachownica := #szachownica) = 1 THEN
                   IF #poz_temp.x = #polozenie_krola.x  AND #poz_temp.y = #polozenie_krola.y  THEN
                       #sprawdz_czy_pion_szach := true;
                   END_IF;
               END_IF;
           END_IF;
       END_IF;
       #poz_temp.x := #pion.pozycja.x;
       #poz_temp.y := #pion.pozycja.y + 1;
       IF "sprawdz_czy_na_szachownicy"(#poz_temp) THEN
           IF "sprawdz_czy_wolne"(pozycja := #poz_temp, szachownica := #szachownica) = 1 THEN
                   IF #poz_temp.x = #polozenie_krola.x  AND #poz_temp.y = #polozenie_krola.y  THEN
                       #sprawdz_czy_pion_szach := true;
                   END_IF;
           END_IF;
       END_IF;
       #poz_temp.x := #pion.pozycja.x - 1;
       #poz_temp.y := #pion.pozycja.y + 1;
       IF "sprawdz_czy_na_szachownicy"(#poz_temp) THEN
           IF "sprawdz_czy_zajete"(pozycja := #poz_temp, szachownica := #szachownica) = 1 THEN
                   IF #poz_temp.x = #polozenie_krola.x  AND #poz_temp.y = #polozenie_krola.y  THEN
                       #sprawdz_czy_pion_szach := true;
                   END_IF;
           END_IF;
       END_IF;
       #poz_temp.x := #pion.pozycja.x + 1;
       #poz_temp.y := #pion.pozycja.y + 1;
       IF "sprawdz_czy_na_szachownicy"(#poz_temp) THEN
           IF "sprawdz_czy_zajete"(pozycja := #poz_temp, szachownica := #szachownica) = 1 THEN
                   IF #poz_temp.x = #polozenie_krola.x  AND #poz_temp.y = #polozenie_krola.y  THEN
                       #sprawdz_czy_pion_szach := true;
                   END_IF;
           END_IF;
       END_IF;
       ELSE
           IF #pion.pozycja.y = 7 THEN
               #poz_temp.x := #pion.pozycja.x;
               #poz_temp.y := #pion.pozycja.y - 2;
               IF "sprawdz_czy_na_szachownicy"(#poz_temp) THEN
                   IF "sprawdz_czy_wolne"(pozycja := #poz_temp, szachownica := #szachownica) = 1 THEN
                   IF #poz_temp.x = #polozenie_krola.x  AND #poz_temp.y = #polozenie_krola.y  THEN
                       #sprawdz_czy_pion_szach := true;
                   END_IF;
                   END_IF;
               END_IF;
           END_IF;
           #poz_temp.x := #pion.pozycja.x;
           #poz_temp.y := #pion.pozycja.y -1;
           IF "sprawdz_czy_na_szachownicy"(#poz_temp) THEN
               IF "sprawdz_czy_wolne"(pozycja := #poz_temp, szachownica := #szachownica) = 1 THEN
                   IF #poz_temp.x = #polozenie_krola.x  AND #poz_temp.y = #polozenie_krola.y  THEN
                       #sprawdz_czy_pion_szach := true;
                   END_IF;
               END_IF;
           END_IF;
           #poz_temp.x := #pion.pozycja.x - 1;
           #poz_temp.y := #pion.pozycja.y - 1;
           IF "sprawdz_czy_na_szachownicy"(#poz_temp) THEN
               IF "sprawdz_czy_zajete"(pozycja := #poz_temp, szachownica := #szachownica) = 2 THEN
                   IF #poz_temp.x = #polozenie_krola.x  AND #poz_temp.y = #polozenie_krola.y  THEN
                       #sprawdz_czy_pion_szach := true;
                   END_IF;
               END_IF;
           END_IF;
           #poz_temp.x := #pion.pozycja.x + 1;
           #poz_temp.y := #pion.pozycja.y - 1;
           IF "sprawdz_czy_na_szachownicy"(#poz_temp) THEN
               IF "sprawdz_czy_zajete"(pozycja := #poz_temp, szachownica := #szachownica) = 2 THEN
                   IF #poz_temp.x = #polozenie_krola.x  AND #poz_temp.y = #polozenie_krola.y  THEN
                       #sprawdz_czy_pion_szach := true;
                   END_IF;
               END_IF;
           END_IF;
   END_IF;
END_FUNCTION

FUNCTION "sprawdz_czy_skoczek_szach" : Bool   // FC19, SCL
{ S7_Optimized_Access := 'TRUE' }
VERSION : 0.1
   VAR_INPUT
      szachownica : "Szachownica";
      polozenie_krola : "Pozycja";
   END_VAR
   VAR_IN_OUT
      skoczek : "Figura";
   END_VAR
   VAR_TEMP
      poz_temp : "Pozycja";
      indeks_mozliwych_ruchow : Int;
   END_VAR
BEGIN

   #sprawdz_czy_skoczek_szach := false;
   IF #skoczek.kolor = 1 THEN
       // ruchy skoczka bialego we wszystkich kierunkach
       #poz_temp.x := #skoczek.pozycja.x + 2;
       #poz_temp.y := #skoczek.pozycja.y + 1;
       IF "sprawdz_czy_na_szachownicy"(#poz_temp) = true THEN
           IF "sprawdz_czy_wolne"(pozycja := #poz_temp, szachownica := #szachownica) = true THEN
               IF #poz_temp.x = #polozenie_krola.x AND #poz_temp.y = #polozenie_krola.y THEN
                   #sprawdz_czy_skoczek_szach := true;
               END_IF;
           ELSIF "sprawdz_czy_zajete"(pozycja := #poz_temp, szachownica := #szachownica) = 1 THEN
               IF #poz_temp.x = #polozenie_krola.x AND #poz_temp.y = #polozenie_krola.y THEN
                   #sprawdz_czy_skoczek_szach := true;
               END_IF;
           END_IF;
       END_IF;
       #poz_temp.x := #skoczek.pozycja.x + 2;
       #poz_temp.y := #skoczek.pozycja.y - 1;
       IF "sprawdz_czy_na_szachownicy"(#poz_temp) = true THEN
           IF "sprawdz_czy_wolne"(pozycja := #poz_temp, szachownica := #szachownica) = true THEN
                   IF #poz_temp.x = #polozenie_krola.x  AND #poz_temp.y = #polozenie_krola.y  THEN
                       #sprawdz_czy_skoczek_szach := true;
                   END_IF;
           ELSIF "sprawdz_czy_zajete"(pozycja := #poz_temp, szachownica := #szachownica) = 1 THEN
                   IF #poz_temp.x = #polozenie_krola.x  AND #poz_temp.y = #polozenie_krola.y  THEN
                       #sprawdz_czy_skoczek_szach := true;
                   END_IF;
           END_IF;
       END_IF;
       #poz_temp.x := #skoczek.pozycja.x - 2;
       #poz_temp.y := #skoczek.pozycja.y + 1;
       IF "sprawdz_czy_na_szachownicy"(#poz_temp) = true THEN
           IF "sprawdz_czy_wolne"(pozycja := #poz_temp, szachownica := #szachownica) = true THEN
                   IF #poz_temp.x = #polozenie_krola.x  AND #poz_temp.y = #polozenie_krola.y  THEN
                       #sprawdz_czy_skoczek_szach := true;
                   END_IF;
           ELSIF "sprawdz_czy_zajete"(pozycja := #poz_temp, szachownica := #szachownica) = 1 THEN
                   IF #poz_temp.x = #polozenie_krola.x  AND #poz_temp.y = #polozenie_krola.y  THEN
                       #sprawdz_czy_skoczek_szach := true;
                   END_IF;
           END_IF;
       END_IF;
       #poz_temp.x := #skoczek.pozycja.x - 2;
       #poz_temp.y := #skoczek.pozycja.y - 1;
       IF "sprawdz_czy_na_szachownicy"(#poz_temp) = true THEN
           IF "sprawdz_czy_wolne"(pozycja := #poz_temp, szachownica := #szachownica) = true THEN
                   IF #poz_temp.x = #polozenie_krola.x  AND #poz_temp.y = #polozenie_krola.y  THEN
                       #sprawdz_czy_skoczek_szach := true;
                   END_IF;
           ELSIF "sprawdz_czy_zajete"(pozycja := #poz_temp, szachownica := #szachownica) = 1 THEN
                   IF #poz_temp.x = #polozenie_krola.x  AND #poz_temp.y = #polozenie_krola.y  THEN
                       #sprawdz_czy_skoczek_szach := true;
                   END_IF;
           END_IF;
       END_IF;
       #poz_temp.x := #skoczek.pozycja.x + 1;
       #poz_temp.y := #skoczek.pozycja.y + 2;
       IF "sprawdz_czy_na_szachownicy"(#poz_temp) = true THEN
           IF "sprawdz_czy_wolne"(pozycja := #poz_temp, szachownica := #szachownica) = true THEN
                   IF #poz_temp.x = #polozenie_krola.x  AND #poz_temp.y = #polozenie_krola.y  THEN
                       #sprawdz_czy_skoczek_szach := true;
                   END_IF;
           ELSIF "sprawdz_czy_zajete"(pozycja := #poz_temp, szachownica := #szachownica) = 1 THEN
                   IF #poz_temp.x = #polozenie_krola.x  AND #poz_temp.y = #polozenie_krola.y  THEN
                       #sprawdz_czy_skoczek_szach := true;
                   END_IF;
           END_IF;
       END_IF;
       #poz_temp.x := #skoczek.pozycja.x - 1;
       #poz_temp.y := #skoczek.pozycja.y + 2;
       IF "sprawdz_czy_na_szachownicy"(#poz_temp) = true THEN
           IF "sprawdz_czy_wolne"(pozycja := #poz_temp, szachownica := #szachownica) = true THEN
                   IF #poz_temp.x = #polozenie_krola.x  AND #poz_temp.y = #polozenie_krola.y  THEN
                       #sprawdz_czy_skoczek_szach := true;
                   END_IF;
           ELSIF "sprawdz_czy_zajete"(pozycja := #poz_temp, szachownica := #szachownica) = 1 THEN
                   IF #poz_temp.x = #polozenie_krola.x  AND #poz_temp.y = #polozenie_krola.y  THEN
                       #sprawdz_czy_skoczek_szach := true;
                   END_IF;
           END_IF;
       END_IF;
       #poz_temp.x := #skoczek.pozycja.x + 1;
       #poz_temp.y := #skoczek.pozycja.y - 2;
       IF "sprawdz_czy_na_szachownicy"(#poz_temp) = true THEN
           IF "sprawdz_czy_wolne"(pozycja := #poz_temp, szachownica := #szachownica) = true THEN
                   IF #poz_temp.x = #polozenie_krola.x  AND #poz_temp.y = #polozenie_krola.y  THEN
                       #sprawdz_czy_skoczek_szach := true;
                   END_IF;
           ELSIF "sprawdz_czy_zajete"(pozycja := #poz_temp, szachownica := #szachownica) = 1 THEN
                   IF #poz_temp.x = #polozenie_krola.x  AND #poz_temp.y = #polozenie_krola.y  THEN
                       #sprawdz_czy_skoczek_szach := true;
                   END_IF;
           END_IF;
       END_IF;
       #poz_temp.x := #skoczek.pozycja.x - 1;
       #poz_temp.y := #skoczek.pozycja.y - 2;
       IF "sprawdz_czy_na_szachownicy"(#poz_temp) = true THEN
           IF "sprawdz_czy_wolne"(pozycja := #poz_temp, szachownica := #szachownica) = true THEN
                   IF #poz_temp.x = #polozenie_krola.x  AND #poz_temp.y = #polozenie_krola.y  THEN
                       #sprawdz_czy_skoczek_szach := true;
                   END_IF;
           ELSIF "sprawdz_czy_zajete"(pozycja := #poz_temp, szachownica := #szachownica) = 1 THEN
                   IF #poz_temp.x = #polozenie_krola.x  AND #poz_temp.y = #polozenie_krola.y  THEN
                       #sprawdz_czy_skoczek_szach := true;
                   END_IF;
           END_IF;
       END_IF;




   ELSE
       // ruchy skoczka czarnego we wszystkich kierunkach
       #poz_temp.x := #skoczek.pozycja.x + 2;
       #poz_temp.y := #skoczek.pozycja.y + 1;
       IF "sprawdz_czy_na_szachownicy"(#poz_temp) = true THEN
           IF "sprawdz_czy_wolne"(pozycja := #poz_temp, szachownica := #szachownica) = true THEN
                   IF #poz_temp.x = #polozenie_krola.x  AND #poz_temp.y = #polozenie_krola.y  THEN
                       #sprawdz_czy_skoczek_szach := true;
                   END_IF;
           ELSIF "sprawdz_czy_zajete"(pozycja := #poz_temp, szachownica := #szachownica) = 2 THEN
                   IF #poz_temp.x = #polozenie_krola.x  AND #poz_temp.y = #polozenie_krola.y  THEN
                       #sprawdz_czy_skoczek_szach := true;
                   END_IF;
           END_IF;
       END_IF;
       #poz_temp.x := #skoczek.pozycja.x + 2;
       #poz_temp.y := #skoczek.pozycja.y - 1;
       IF "sprawdz_czy_na_szachownicy"(#poz_temp) = true THEN
           IF "sprawdz_czy_wolne"(pozycja := #poz_temp, szachownica := #szachownica) = true THEN
                   IF #poz_temp.x = #polozenie_krola.x  AND #poz_temp.y = #polozenie_krola.y  THEN
                       #sprawdz_czy_skoczek_szach := true;
                   END_IF;
           ELSIF "sprawdz_czy_zajete"(pozycja := #poz_temp, szachownica := #szachownica) = 2 THEN
                   IF #poz_temp.x = #polozenie_krola.x  AND #poz_temp.y = #polozenie_krola.y  THEN
                       #sprawdz_czy_skoczek_szach := true;
                   END_IF;
           END_IF;
       END_IF;
       #poz_temp.x := #skoczek.pozycja.x - 2;
       #poz_temp.y := #skoczek.pozycja.y + 1;
       IF "sprawdz_czy_na_szachownicy"(#poz_temp) = true THEN
           IF "sprawdz_czy_wolne"(pozycja := #poz_temp, szachownica := #szachownica) = true THEN
                   IF #poz_temp.x = #polozenie_krola.x  AND #poz_temp.y = #polozenie_krola.y  THEN
                       #sprawdz_czy_skoczek_szach := true;
                   END_IF;
           ELSIF "sprawdz_czy_zajete"(pozycja := #poz_temp, szachownica := #szachownica) = 2 THEN
                   IF #poz_temp.x = #polozenie_krola.x  AND #poz_temp.y = #polozenie_krola.y  THEN
                       #sprawdz_czy_skoczek_szach := true;
                   END_IF;
           END_IF;
       END_IF;
       #poz_temp.x := #skoczek.pozycja.x - 2;
       #poz_temp.y := #skoczek.pozycja.y - 1;
       IF "sprawdz_czy_na_szachownicy"(#poz_temp) = true THEN
           IF "sprawdz_czy_wolne"(pozycja := #poz_temp, szachownica := #szachownica) = true THEN
                   IF #poz_temp.x = #polozenie_krola.x  AND #poz_temp.y = #polozenie_krola.y  THEN
                       #sprawdz_czy_skoczek_szach := true;
                   END_IF;
           ELSIF "sprawdz_czy_zajete"(pozycja := #poz_temp, szachownica := #szachownica) = 2 THEN
                   IF #poz_temp.x = #polozenie_krola.x  AND #poz_temp.y = #polozenie_krola.y  THEN
                       #sprawdz_czy_skoczek_szach := true;
                   END_IF;
           END_IF;
       END_IF;
       #poz_temp.x := #skoczek.pozycja.x + 1;
       #poz_temp.y := #skoczek.pozycja.y + 2;
       IF "sprawdz_czy_na_szachownicy"(#poz_temp) = true THEN
           IF "sprawdz_czy_wolne"(pozycja := #poz_temp, szachownica := #szachownica) = true THEN
                   IF #poz_temp.x = #polozenie_krola.x  AND #poz_temp.y = #polozenie_krola.y  THEN
                       #sprawdz_czy_skoczek_szach := true;
                   END_IF;
           ELSIF "sprawdz_czy_zajete"(pozycja := #poz_temp, szachownica := #szachownica) = 2 THEN
                    IF #poz_temp.x = #polozenie_krola.x  AND #poz_temp.y = #polozenie_krola.y  THEN
                       #sprawdz_czy_skoczek_szach := true;
                   END_IF;
           END_IF;
       END_IF;
       #poz_temp.x := #skoczek.pozycja.x - 1;
       #poz_temp.y := #skoczek.pozycja.y + 2;
       IF "sprawdz_czy_na_szachownicy"(#poz_temp) = true THEN
           IF "sprawdz_czy_wolne"(pozycja := #poz_temp, szachownica := #szachownica) = true THEN
                   IF #poz_temp.x = #polozenie_krola.x  AND #poz_temp.y = #polozenie_krola.y  THEN
                       #sprawdz_czy_skoczek_szach := true;
                   END_IF;
           ELSIF "sprawdz_czy_zajete"(pozycja := #poz_temp, szachownica := #szachownica) = 2 THEN
                   IF #poz_temp.x = #polozenie_krola.x  AND #poz_temp.y = #polozenie_krola.y  THEN
                       #sprawdz_czy_skoczek_szach := true;
                   END_IF;
           END_IF;
       END_IF;
       #poz_temp.x := #skoczek.pozycja.x + 1;
       #poz_temp.y := #skoczek.pozycja.y - 2;
       IF "sprawdz_czy_na_szachownicy"(#poz_temp) = true THEN
           IF "sprawdz_czy_wolne"(pozycja := #poz_temp, szachownica := #szachownica) = true THEN
                   IF #poz_temp.x = #polozenie_krola.x  AND #poz_temp.y = #polozenie_krola.y  THEN
                       #sprawdz_czy_skoczek_szach := true;
                   END_IF;
           ELSIF "sprawdz_czy_zajete"(pozycja := #poz_temp, szachownica := #szachownica) = 2 THEN
                   IF #poz_temp.x = #polozenie_krola.x  AND #poz_temp.y = #polozenie_krola.y  THEN
                       #sprawdz_czy_skoczek_szach := true;
                   END_IF;
           END_IF;
       END_IF;
       #poz_temp.x := #skoczek.pozycja.x - 1;
       #poz_temp.y := #skoczek.pozycja.y - 2;
       IF "sprawdz_czy_na_szachownicy"(#poz_temp) = true THEN
           IF "sprawdz_czy_wolne"(pozycja := #poz_temp, szachownica := #szachownica) = true THEN
                   IF #poz_temp.x = #polozenie_krola.x  AND #poz_temp.y = #polozenie_krola.y  THEN
                       #sprawdz_czy_skoczek_szach := true;
                   END_IF;
           ELSIF "sprawdz_czy_zajete"(pozycja := #poz_temp, szachownica := #szachownica) = 2 THEN
                   IF #poz_temp.x = #polozenie_krola.x  AND #poz_temp.y = #polozenie_krola.y  THEN
                       #sprawdz_czy_skoczek_szach := true;
                   END_IF;
           END_IF;
       END_IF;

   END_IF;
END_FUNCTION

FUNCTION "sprawdz_czy_goniec_szach" : Bool   // FC20, SCL
{ S7_Optimized_Access := 'TRUE' }
VERSION : 0.1
   VAR_INPUT
      szachownica : "Szachownica";
      polozenie_krola : "Pozycja";
   END_VAR
   VAR_IN_OUT
      goniec : "Figura";
   END_VAR
   VAR_TEMP
      poz_temp : "Pozycja";
      indeks_mozliwych_ruchow : Int;
      wykonuj_petle : Bool;
   END_VAR
BEGIN
   #poz_temp := #goniec.pozycja;
   #sprawdz_czy_goniec_szach := false;
   IF #goniec.kolor = 1 THEN
       #wykonuj_petle := TRUE;
       #poz_temp := #goniec.pozycja;
       WHILE #wykonuj_petle DO
           #poz_temp.x += 1;
           #poz_temp.y += 1;
           IF "sprawdz_czy_na_szachownicy"(#poz_temp) = true THEN
               IF "sprawdz_czy_wolne"(pozycja := #poz_temp, szachownica := #szachownica) = true THEN
                   IF #poz_temp.x = #polozenie_krola.x AND #poz_temp.y = #polozenie_krola.y  THEN
                       #sprawdz_czy_goniec_szach := true;
                   END_IF;
               ELSIF "sprawdz_czy_zajete"(pozycja := #poz_temp, szachownica := #szachownica) = 1 THEN
                   IF #poz_temp.x = #polozenie_krola.x AND #poz_temp.y = #polozenie_krola.y  THEN
                       #sprawdz_czy_goniec_szach := true;
                   ELSE
                       #wykonuj_petle := false;
                   END_IF;
               ELSE
                   #wykonuj_petle := false;
               END_IF;
           ELSE
               #wykonuj_petle := false;
           END_IF;
       END_WHILE;
       #wykonuj_petle := TRUE;
       #poz_temp := #goniec.pozycja;
       WHILE #wykonuj_petle DO
           #poz_temp.x += 1;
           #poz_temp.y -= 1;
           IF "sprawdz_czy_na_szachownicy"(#poz_temp) = true THEN
               IF "sprawdz_czy_wolne"(pozycja := #poz_temp, szachownica := #szachownica) = true THEN
                   IF #poz_temp.x = #polozenie_krola.x AND #poz_temp.y = #polozenie_krola.y  THEN
                       #sprawdz_czy_goniec_szach := true;
                   END_IF;
               ELSIF "sprawdz_czy_zajete"(pozycja := #poz_temp, szachownica := #szachownica) = 1 THEN
                   IF #poz_temp.x = #polozenie_krola.x AND #poz_temp.y = #polozenie_krola.y  THEN
                       #sprawdz_czy_goniec_szach := true;
                   ELSE
                       #wykonuj_petle := false;
                   END_IF;
               ELSE
                   #wykonuj_petle := false;
               END_IF;
           ELSE
               #wykonuj_petle := false;
           END_IF;
       END_WHILE;
       #wykonuj_petle := TRUE;
       #poz_temp := #goniec.pozycja;
       WHILE #wykonuj_petle DO
           #poz_temp.x -= 1;
           #poz_temp.y += 1;
           IF "sprawdz_czy_na_szachownicy"(#poz_temp) = true THEN
               IF "sprawdz_czy_wolne"(pozycja := #poz_temp, szachownica := #szachownica) = true THEN
                   IF #poz_temp.x = #polozenie_krola.x AND #poz_temp.y = #polozenie_krola.y  THEN
                       #sprawdz_czy_goniec_szach := true;
                   END_IF;
               ELSIF "sprawdz_czy_zajete"(pozycja := #poz_temp, szachownica := #szachownica) = 1 THEN
                   IF #poz_temp.x = #polozenie_krola.x AND #poz_temp.y = #polozenie_krola.y  THEN
                       #sprawdz_czy_goniec_szach := true;
                   ELSE
                       #wykonuj_petle := false;
                   END_IF;
               ELSE
                   #wykonuj_petle := false;
               END_IF;
           ELSE
               #wykonuj_petle := false;
           END_IF;
       END_WHILE;
       #wykonuj_petle := TRUE;
       #poz_temp := #goniec.pozycja;
       WHILE #wykonuj_petle DO
           #poz_temp.x -= 1;
           #poz_temp.y -= 1;
           IF "sprawdz_czy_na_szachownicy"(#poz_temp) = true THEN
               IF "sprawdz_czy_wolne"(pozycja := #poz_temp, szachownica := #szachownica) = true THEN
                   IF #poz_temp.x = #polozenie_krola.x AND #poz_temp.y = #polozenie_krola.y  THEN
                       #sprawdz_czy_goniec_szach := true;
                   END_IF;
               ELSIF "sprawdz_czy_zajete"(pozycja := #poz_temp, szachownica := #szachownica) = 1 THEN
                   IF #poz_temp.x = #polozenie_krola.x AND #poz_temp.y = #polozenie_krola.y  THEN
                       #sprawdz_czy_goniec_szach := true;
                   ELSE
                       #wykonuj_petle := false;
                   END_IF;
               ELSE
                   #wykonuj_petle := false;
               END_IF;
           ELSE
               #wykonuj_petle := false;
           END_IF;
       END_WHILE;


   ELSE
       #wykonuj_petle := TRUE;
       #poz_temp := #goniec.pozycja;
       WHILE #wykonuj_petle DO
           #poz_temp.x += 1;
           #poz_temp.y += 1;
           IF "sprawdz_czy_na_szachownicy"(#poz_temp) = true THEN
               IF "sprawdz_czy_wolne"(pozycja := #poz_temp, szachownica := #szachownica) = true THEN
                   IF #poz_temp.x = #polozenie_krola.x AND #poz_temp.y = #polozenie_krola.y  THEN
                       #sprawdz_czy_goniec_szach := true;
                   END_IF;
               ELSIF "sprawdz_czy_zajete"(pozycja := #poz_temp, szachownica := #szachownica) = 2 THEN
                   IF #poz_temp.x = #polozenie_krola.x AND #poz_temp.y = #polozenie_krola.y  THEN
                       #sprawdz_czy_goniec_szach := true;
                   ELSE
                       #wykonuj_petle := false;
                   END_IF;
               ELSE
                   #wykonuj_petle := false;
               END_IF;
           ELSE
               #wykonuj_petle := false;
           END_IF;
       END_WHILE;
       #wykonuj_petle := TRUE;
       #poz_temp := #goniec.pozycja;
       WHILE #wykonuj_petle DO
           #poz_temp.x += 1;
           #poz_temp.y -= 1;
           IF "sprawdz_czy_na_szachownicy"(#poz_temp) = true THEN
               IF "sprawdz_czy_wolne"(pozycja := #poz_temp, szachownica := #szachownica) = true THEN
                   IF #poz_temp.x = #polozenie_krola.x AND #poz_temp.y = #polozenie_krola.y  THEN
                       #sprawdz_czy_goniec_szach := true;
                   END_IF;
               ELSIF "sprawdz_czy_zajete"(pozycja := #poz_temp, szachownica := #szachownica) = 2 THEN
                   IF #poz_temp.x = #polozenie_krola.x AND #poz_temp.y = #polozenie_krola.y  THEN
                       #sprawdz_czy_goniec_szach := true;
                   ELSE
                       #wykonuj_petle := false;
                   END_IF;
               ELSE
                   #wykonuj_petle := false;
               END_IF;
           ELSE
               #wykonuj_petle := false;
           END_IF;
       END_WHILE;
       #wykonuj_petle := TRUE;
       #poz_temp := #goniec.pozycja;
       WHILE #wykonuj_petle DO
           #poz_temp.x -= 1;
           #poz_temp.y += 1;
           IF "sprawdz_czy_na_szachownicy"(#poz_temp) = true THEN
               IF "sprawdz_czy_wolne"(pozycja := #poz_temp, szachownica := #szachownica) = true THEN
                   IF #poz_temp.x = #polozenie_krola.x AND #poz_temp.y = #polozenie_krola.y  THEN
                       #sprawdz_czy_goniec_szach := true;
                   END_IF;
               ELSIF "sprawdz_czy_zajete"(pozycja := #poz_temp, szachownica := #szachownica) = 2 THEN
                   IF #poz_temp.x = #polozenie_krola.x AND #poz_temp.y = #polozenie_krola.y  THEN
                       #sprawdz_czy_goniec_szach := true;
                   ELSE
                       #wykonuj_petle := false;
                   END_IF;
               ELSE
                   #wykonuj_petle := false;
               END_IF;
           ELSE
               #wykonuj_petle := false;
           END_IF;
       END_WHILE;
       #wykonuj_petle := TRUE;
       #poz_temp := #goniec.pozycja;
       WHILE #wykonuj_petle DO
           #poz_temp.x -= 1;
           #poz_temp.y -= 1;
           IF "sprawdz_czy_na_szachownicy"(#poz_temp) = true THEN
               IF "sprawdz_czy_wolne"(pozycja := #poz_temp, szachownica := #szachownica) = true THEN
                   IF #poz_temp.x = #polozenie_krola.x AND #poz_temp.y = #polozenie_krola.y  THEN
                       #sprawdz_czy_goniec_szach := true;
                   END_IF;
               ELSIF "sprawdz_czy_zajete"(pozycja := #poz_temp, szachownica := #szachownica) = 2 THEN
                   IF #poz_temp.x = #polozenie_krola.x AND #poz_temp.y = #polozenie_krola.y  THEN
                       #sprawdz_czy_goniec_szach := true;
                   ELSE
                       #wykonuj_petle := false;
                   END_IF;
               ELSE
                   #wykonuj_petle := false;
               END_IF;
           ELSE
               #wykonuj_petle := false;
           END_IF;
       END_WHILE;
   END_IF;
END_FUNCTION

FUNCTION "sprawdz_czy_wieza_szach" : Bool   // FC21, SCL
{ S7_Optimized_Access := 'TRUE' }
VERSION : 0.1
   VAR_INPUT
      szachownica : "Szachownica";
      polozenie_krola : "Pozycja";
   END_VAR
   VAR_IN_OUT
      wieza : "Figura";
   END_VAR
   VAR_TEMP
      poz_temp : "Pozycja";
      wykonuj_petle : Bool;
      indeks_mozliwych_ruchow : Int;
   END_VAR
BEGIN
   #indeks_mozliwych_ruchow := 0;
   #sprawdz_czy_wieza_szach := false;

   IF #wieza.kolor = 1 THEN
       // ruch białych 
       // 
       //ruch poziomo i pionowo
       #wykonuj_petle := TRUE;
       #poz_temp := #wieza.pozycja;
       WHILE #wykonuj_petle DO
           #poz_temp.x += 1;
           #poz_temp.y += 0;
           IF "sprawdz_czy_na_szachownicy"(#poz_temp) = true THEN
               IF "sprawdz_czy_wolne"(pozycja := #poz_temp, szachownica := #szachownica) = true THEN
               IF #poz_temp.x = #polozenie_krola.x AND #poz_temp.y = #polozenie_krola.y THEN
                   #sprawdz_czy_wieza_szach := true;
               END_IF;
               ELSIF "sprawdz_czy_zajete"(pozycja := #poz_temp, szachownica := #szachownica) = 1 THEN
               IF #poz_temp.x = #polozenie_krola.x AND #poz_temp.y = #polozenie_krola.y THEN
                   #sprawdz_czy_wieza_szach := true;
               ELSE
                   #wykonuj_petle := false;
               END_IF;
           ELSE
               #wykonuj_petle := false;
               END_IF;
           ELSE
               #wykonuj_petle := false;
           END_IF;
       END_WHILE;
       #wykonuj_petle := TRUE;
       #poz_temp := #wieza.pozycja;
       WHILE #wykonuj_petle DO
           #poz_temp.x += 0;
           #poz_temp.y += 1;
           IF "sprawdz_czy_na_szachownicy"(#poz_temp) = true THEN
               IF "sprawdz_czy_wolne"(pozycja := #poz_temp, szachownica := #szachownica) = true THEN
               IF #poz_temp.x = #polozenie_krola.x AND #poz_temp.y = #polozenie_krola.y THEN
                   #sprawdz_czy_wieza_szach := true;
               END_IF;
               ELSIF "sprawdz_czy_zajete"(pozycja := #poz_temp, szachownica := #szachownica) = 1 THEN
               IF #poz_temp.x = #polozenie_krola.x AND #poz_temp.y = #polozenie_krola.y THEN
                   #sprawdz_czy_wieza_szach := true;
               ELSE
                   #wykonuj_petle := false;
               END_IF;
           ELSE
               #wykonuj_petle := false;
               END_IF;
           ELSE
               #wykonuj_petle := false;
           END_IF;
       END_WHILE;
       #wykonuj_petle := TRUE;
       #poz_temp := #wieza.pozycja;
       WHILE #wykonuj_petle DO
           #poz_temp.x += -1;
           #poz_temp.y += 0;
           IF "sprawdz_czy_na_szachownicy"(#poz_temp) = true THEN
               IF "sprawdz_czy_wolne"(pozycja := #poz_temp, szachownica := #szachownica) = true THEN
               IF #poz_temp.x = #polozenie_krola.x AND #poz_temp.y = #polozenie_krola.y THEN
                   #sprawdz_czy_wieza_szach := true;
               END_IF;
               ELSIF "sprawdz_czy_zajete"(pozycja := #poz_temp, szachownica := #szachownica) = 1 THEN
               IF #poz_temp.x = #polozenie_krola.x AND #poz_temp.y = #polozenie_krola.y THEN
                   #sprawdz_czy_wieza_szach := true;
               ELSE
                   #wykonuj_petle := false;
               END_IF;
           ELSE
               #wykonuj_petle := false;
               END_IF;
           ELSE
               #wykonuj_petle := false;
           END_IF;
       END_WHILE;
       #wykonuj_petle := TRUE;
       #poz_temp := #wieza.pozycja;
       WHILE #wykonuj_petle DO
           #poz_temp.x += 0;
           #poz_temp.y += -1;
           IF "sprawdz_czy_na_szachownicy"(#poz_temp) = true THEN
               IF "sprawdz_czy_wolne"(pozycja := #poz_temp, szachownica := #szachownica) = true THEN
               IF #poz_temp.x = #polozenie_krola.x AND #poz_temp.y = #polozenie_krola.y THEN
                   #sprawdz_czy_wieza_szach := true;
               END_IF;
               ELSIF "sprawdz_czy_zajete"(pozycja := #poz_temp, szachownica := #szachownica) = 1 THEN
               IF #poz_temp.x = #polozenie_krola.x AND #poz_temp.y = #polozenie_krola.y THEN
                   #sprawdz_czy_wieza_szach := true;
               ELSE
                   #wykonuj_petle := false;
               END_IF;
           ELSE
               #wykonuj_petle := false;
               END_IF;
           ELSE
               #wykonuj_petle := false;
           END_IF;
       END_WHILE;


   ELSE
       //ruch czarnych
       //
       //ruch poziomo i pionowo
       #wykonuj_petle := TRUE;
       #poz_temp := #wieza.pozycja;
       WHILE #wykonuj_petle DO
           #poz_temp.x += 1;
           #poz_temp.y += 0;
           IF "sprawdz_czy_na_szachownicy"(#poz_temp) = true THEN
               IF "sprawdz_czy_wolne"(pozycja := #poz_temp, szachownica := #szachownica) = true THEN
               IF #poz_temp.x = #polozenie_krola.x AND #poz_temp.y = #polozenie_krola.y THEN
                   #sprawdz_czy_wieza_szach := true;
               END_IF;
               ELSIF "sprawdz_czy_zajete"(pozycja := #poz_temp, szachownica := #szachownica) = 2 THEN
               IF #poz_temp.x = #polozenie_krola.x AND #poz_temp.y = #polozenie_krola.y THEN
                   #sprawdz_czy_wieza_szach := true;
               ELSE
                   #wykonuj_petle := false;
               END_IF;
           ELSE
               #wykonuj_petle := false;
               END_IF;
           ELSE
               #wykonuj_petle := false;
           END_IF;
       END_WHILE;
       #wykonuj_petle := TRUE;
       #poz_temp := #wieza.pozycja;
       WHILE #wykonuj_petle DO
           #poz_temp.x += 0;
           #poz_temp.y += 1;
           IF "sprawdz_czy_na_szachownicy"(#poz_temp) = true THEN
               IF "sprawdz_czy_wolne"(pozycja := #poz_temp, szachownica := #szachownica) = true THEN
               IF #poz_temp.x = #polozenie_krola.x AND #poz_temp.y = #polozenie_krola.y THEN
                   #sprawdz_czy_wieza_szach := true;
               END_IF;
               ELSIF "sprawdz_czy_zajete"(pozycja := #poz_temp, szachownica := #szachownica) = 2 THEN
               IF #poz_temp.x = #polozenie_krola.x AND #poz_temp.y = #polozenie_krola.y THEN
                   #sprawdz_czy_wieza_szach := true;
               ELSE
                   #wykonuj_petle := false;
               END_IF;
           ELSE
               #wykonuj_petle := false;
               END_IF;
           ELSE
               #wykonuj_petle := false;
           END_IF;
       END_WHILE;
       #wykonuj_petle := TRUE;
       #poz_temp := #wieza.pozycja;
       WHILE #wykonuj_petle DO
           #poz_temp.x += -1;
           #poz_temp.y += 0;
           IF "sprawdz_czy_na_szachownicy"(#poz_temp) = true THEN
               IF "sprawdz_czy_wolne"(pozycja := #poz_temp, szachownica := #szachownica) = true THEN
               IF #poz_temp.x = #polozenie_krola.x AND #poz_temp.y = #polozenie_krola.y THEN
                   #sprawdz_czy_wieza_szach := true;
               END_IF;
               ELSIF "sprawdz_czy_zajete"(pozycja := #poz_temp, szachownica := #szachownica) = 2 THEN
               IF #poz_temp.x = #polozenie_krola.x AND #poz_temp.y = #polozenie_krola.y THEN
                   #sprawdz_czy_wieza_szach := true;
               ELSE
                   #wykonuj_petle := false;
               END_IF;
           ELSE
               #wykonuj_petle := false;
               END_IF;
           ELSE
               #wykonuj_petle := false;
           END_IF;
       END_WHILE;
       #wykonuj_petle := TRUE;
       #poz_temp := #wieza.pozycja;
       WHILE #wykonuj_petle DO
           #poz_temp.x += 0;
           #poz_temp.y += -1;
           IF "sprawdz_czy_na_szachownicy"(#poz_temp) = true THEN
               IF "sprawdz_czy_wolne"(pozycja := #poz_temp, szachownica := #szachownica) = true THEN
               IF #poz_temp.x = #polozenie_krola.x AND #poz_temp.y = #polozenie_krola.y THEN
                   #sprawdz_czy_wieza_szach := true;
               END_IF;
               ELSIF "sprawdz_czy_zajete"(pozycja := #poz_temp, szachownica := #szachownica) = 2 THEN
               IF #poz_temp.x = #polozenie_krola.x AND #poz_temp.y = #polozenie_krola.y THEN
                   #sprawdz_czy_wieza_szach := true;
               ELSE
                   #wykonuj_petle := false;
               END_IF;
           ELSE
               #wykonuj_petle := false;
               END_IF;
           ELSE
               #wykonuj_petle := false;
           END_IF;
       END_WHILE;
   END_IF;
END_FUNCTION

FUNCTION "sprawdz_czy_krol_szach" : Bool   // FC22, SCL
{ S7_Optimized_Access := 'TRUE' }
VERSION : 0.1
   VAR_INPUT
      szachownica : "Szachownica";
      polozenie_krola : "Pozycja";
   END_VAR
   VAR_IN_OUT
      krol : "Figura";
   END_VAR
   VAR_TEMP
      poz_temp : "Pozycja";
      indeks_mozliwych_ruchow : Int;
   END_VAR
BEGIN
   #indeks_mozliwych_ruchow := 0;
   #sprawdz_czy_krol_szach := false;
   IF #krol.kolor = 1 THEN
       // ruchy króla bialego we wszystkich kierunkach
       #poz_temp.x := #krol.pozycja.x;
       #poz_temp.y := #krol.pozycja.y + 1;
       IF "sprawdz_czy_na_szachownicy"(#poz_temp) = true THEN
           IF "sprawdz_czy_wolne"(pozycja := #poz_temp, szachownica := #szachownica) = true THEN
                   IF #poz_temp.x = #polozenie_krola.x  AND #poz_temp.y = #polozenie_krola.y  THEN
                       #sprawdz_czy_krol_szach := true;
                   END_IF;
           ELSIF "sprawdz_czy_zajete"(pozycja := #poz_temp, szachownica := #szachownica) = 1 THEN
                   IF #poz_temp.x = #polozenie_krola.x  AND #poz_temp.y = #polozenie_krola.y  THEN
                       #sprawdz_czy_krol_szach := true;
                   END_IF;
           END_IF;
       END_IF;
       #poz_temp.x := #krol.pozycja.x + 1;
       #poz_temp.y := #krol.pozycja.y + 1;
       IF "sprawdz_czy_na_szachownicy"(#poz_temp) = true THEN
           IF "sprawdz_czy_wolne"(pozycja := #poz_temp, szachownica := #szachownica) = true THEN
                   IF #poz_temp.x = #polozenie_krola.x  AND #poz_temp.y = #polozenie_krola.y  THEN
                       #sprawdz_czy_krol_szach := true;
                   END_IF;
           ELSIF "sprawdz_czy_zajete"(pozycja := #poz_temp, szachownica := #szachownica) = 1 THEN
                   IF #poz_temp.x = #polozenie_krola.x  AND #poz_temp.y = #polozenie_krola.y  THEN
                       #sprawdz_czy_krol_szach := true;
                   END_IF;
           END_IF;
       END_IF;
       #poz_temp.x := #krol.pozycja.x + 1;
       #poz_temp.y := #krol.pozycja.y;
       IF "sprawdz_czy_na_szachownicy"(#poz_temp) = true THEN
           IF "sprawdz_czy_wolne"(pozycja := #poz_temp, szachownica := #szachownica) = true THEN
                   IF #poz_temp.x = #polozenie_krola.x  AND #poz_temp.y = #polozenie_krola.y  THEN
                       #sprawdz_czy_krol_szach := true;
                   END_IF;
           ELSIF "sprawdz_czy_zajete"(pozycja := #poz_temp, szachownica := #szachownica) = 1 THEN
                   IF #poz_temp.x = #polozenie_krola.x  AND #poz_temp.y = #polozenie_krola.y  THEN
                       #sprawdz_czy_krol_szach := true;
                   END_IF;
           END_IF;
       END_IF;
       #poz_temp.x := #krol.pozycja.x + 1;
       #poz_temp.y := #krol.pozycja.y - 1;
       IF "sprawdz_czy_na_szachownicy"(#poz_temp) = true THEN
           IF "sprawdz_czy_wolne"(pozycja := #poz_temp, szachownica := #szachownica) = true THEN
                   IF #poz_temp.x = #polozenie_krola.x  AND #poz_temp.y = #polozenie_krola.y  THEN
                       #sprawdz_czy_krol_szach := true;
                   END_IF;
           ELSIF "sprawdz_czy_zajete"(pozycja := #poz_temp, szachownica := #szachownica) = 1 THEN
                   IF #poz_temp.x = #polozenie_krola.x  AND #poz_temp.y = #polozenie_krola.y  THEN
                       #sprawdz_czy_krol_szach := true;
                   END_IF;
           END_IF;
       END_IF;
       #poz_temp.x := #krol.pozycja.x;
       #poz_temp.y := #krol.pozycja.y - 1;
       IF "sprawdz_czy_na_szachownicy"(#poz_temp) = true THEN
           IF "sprawdz_czy_wolne"(pozycja := #poz_temp, szachownica := #szachownica) = true THEN
                   IF #poz_temp.x = #polozenie_krola.x  AND #poz_temp.y = #polozenie_krola.y  THEN
                       #sprawdz_czy_krol_szach := true;
                   END_IF;
           ELSIF "sprawdz_czy_zajete"(pozycja := #poz_temp, szachownica := #szachownica) = 1 THEN
                   IF #poz_temp.x = #polozenie_krola.x  AND #poz_temp.y = #polozenie_krola.y  THEN
                       #sprawdz_czy_krol_szach := true;
                   END_IF;
           END_IF;
       END_IF;
       #poz_temp.x := #krol.pozycja.x - 1;
       #poz_temp.y := #krol.pozycja.y - 1;
       IF "sprawdz_czy_na_szachownicy"(#poz_temp) = true THEN
           IF "sprawdz_czy_wolne"(pozycja := #poz_temp, szachownica := #szachownica) = true THEN
                   IF #poz_temp.x = #polozenie_krola.x  AND #poz_temp.y = #polozenie_krola.y  THEN
                       #sprawdz_czy_krol_szach := true;
                   END_IF;
           ELSIF "sprawdz_czy_zajete"(pozycja := #poz_temp, szachownica := #szachownica) = 1 THEN
                   IF #poz_temp.x = #polozenie_krola.x  AND #poz_temp.y = #polozenie_krola.y  THEN
                       #sprawdz_czy_krol_szach := true;
                   END_IF;
           END_IF;
       END_IF;
       #poz_temp.x := #krol.pozycja.x - 1;
       #poz_temp.y := #krol.pozycja.y;
       IF "sprawdz_czy_na_szachownicy"(#poz_temp) = true THEN
           IF "sprawdz_czy_wolne"(pozycja := #poz_temp, szachownica := #szachownica) = true THEN
                   IF #poz_temp.x = #polozenie_krola.x  AND #poz_temp.y = #polozenie_krola.y  THEN
                       #sprawdz_czy_krol_szach := true;
                   END_IF;
           ELSIF "sprawdz_czy_zajete"(pozycja := #poz_temp, szachownica := #szachownica) = 1 THEN
                   IF #poz_temp.x = #polozenie_krola.x  AND #poz_temp.y = #polozenie_krola.y  THEN
                       #sprawdz_czy_krol_szach := true;
                   END_IF;
           END_IF;
       END_IF;
       #poz_temp.x := #krol.pozycja.x - 1;
       #poz_temp.y := #krol.pozycja.y + 1;
       IF "sprawdz_czy_na_szachownicy"(#poz_temp) = true THEN
           IF "sprawdz_czy_wolne"(pozycja := #poz_temp, szachownica := #szachownica) = true THEN
                   IF #poz_temp.x = #polozenie_krola.x  AND #poz_temp.y = #polozenie_krola.y  THEN
                       #sprawdz_czy_krol_szach := true;
                   END_IF;
           ELSIF "sprawdz_czy_zajete"(pozycja := #poz_temp, szachownica := #szachownica) = 1 THEN
                   IF #poz_temp.x = #polozenie_krola.x  AND #poz_temp.y = #polozenie_krola.y  THEN
                       #sprawdz_czy_krol_szach := true;
                   END_IF;
           END_IF;
       END_IF;


   ELSE
       // ruchy króla bialego we wszystkich kierunkach
       #poz_temp.x := #krol.pozycja.x;
       #poz_temp.y := #krol.pozycja.y + 1;
       IF "sprawdz_czy_na_szachownicy"(#poz_temp) = true THEN
           IF "sprawdz_czy_wolne"(pozycja := #poz_temp, szachownica := #szachownica) = true THEN
                   IF #poz_temp.x = #polozenie_krola.x  AND #poz_temp.y = #polozenie_krola.y  THEN
                       #sprawdz_czy_krol_szach := true;
                   END_IF;
           ELSIF "sprawdz_czy_zajete"(pozycja := #poz_temp, szachownica := #szachownica) = 2 THEN
                   IF #poz_temp.x = #polozenie_krola.x  AND #poz_temp.y = #polozenie_krola.y  THEN
                       #sprawdz_czy_krol_szach := true;
                   END_IF;
           END_IF;
       END_IF;
       #poz_temp.x := #krol.pozycja.x + 1;
       #poz_temp.y := #krol.pozycja.y + 1;
       IF "sprawdz_czy_na_szachownicy"(#poz_temp) = true THEN
           IF "sprawdz_czy_wolne"(pozycja := #poz_temp, szachownica := #szachownica) = true THEN
                   IF #poz_temp.x = #polozenie_krola.x  AND #poz_temp.y = #polozenie_krola.y  THEN
                       #sprawdz_czy_krol_szach := true;
                   END_IF;
           ELSIF "sprawdz_czy_zajete"(pozycja := #poz_temp, szachownica := #szachownica) = 2 THEN
                   IF #poz_temp.x = #polozenie_krola.x  AND #poz_temp.y = #polozenie_krola.y  THEN
                       #sprawdz_czy_krol_szach := true;
                   END_IF;
           END_IF;
       END_IF;
       #poz_temp.x := #krol.pozycja.x + 1;
       #poz_temp.y := #krol.pozycja.y;
       IF "sprawdz_czy_na_szachownicy"(#poz_temp) = true THEN
           IF "sprawdz_czy_wolne"(pozycja := #poz_temp, szachownica := #szachownica) = true THEN
                   IF #poz_temp.x = #polozenie_krola.x  AND #poz_temp.y = #polozenie_krola.y  THEN
                       #sprawdz_czy_krol_szach := true;
                   END_IF;
           ELSIF "sprawdz_czy_zajete"(pozycja := #poz_temp, szachownica := #szachownica) = 2 THEN
                   IF #poz_temp.x = #polozenie_krola.x  AND #poz_temp.y = #polozenie_krola.y  THEN
                       #sprawdz_czy_krol_szach := true;
                   END_IF;
           END_IF;
       END_IF;
       #poz_temp.x := #krol.pozycja.x + 1;
       #poz_temp.y := #krol.pozycja.y - 1;
       IF "sprawdz_czy_na_szachownicy"(#poz_temp) = true THEN
           IF "sprawdz_czy_wolne"(pozycja := #poz_temp, szachownica := #szachownica) = true THEN
                   IF #poz_temp.x = #polozenie_krola.x  AND #poz_temp.y = #polozenie_krola.y  THEN
                       #sprawdz_czy_krol_szach := true;
                   END_IF;
           ELSIF "sprawdz_czy_zajete"(pozycja := #poz_temp, szachownica := #szachownica) = 2 THEN
                   IF #poz_temp.x = #polozenie_krola.x  AND #poz_temp.y = #polozenie_krola.y  THEN
                       #sprawdz_czy_krol_szach := true;
                   END_IF;
           END_IF;
       END_IF;
       #poz_temp.x := #krol.pozycja.x;
       #poz_temp.y := #krol.pozycja.y - 1;
       IF "sprawdz_czy_na_szachownicy"(#poz_temp) = true THEN
           IF "sprawdz_czy_wolne"(pozycja := #poz_temp, szachownica := #szachownica) = true THEN
                   IF #poz_temp.x = #polozenie_krola.x  AND #poz_temp.y = #polozenie_krola.y  THEN
                       #sprawdz_czy_krol_szach := true;
                   END_IF;
           ELSIF "sprawdz_czy_zajete"(pozycja := #poz_temp, szachownica := #szachownica) = 2 THEN
                   IF #poz_temp.x = #polozenie_krola.x  AND #poz_temp.y = #polozenie_krola.y  THEN
                       #sprawdz_czy_krol_szach := true;
                   END_IF;
           END_IF;
       END_IF;
       #poz_temp.x := #krol.pozycja.x - 1;
       #poz_temp.y := #krol.pozycja.y - 1;
       IF "sprawdz_czy_na_szachownicy"(#poz_temp) = true THEN
           IF "sprawdz_czy_wolne"(pozycja := #poz_temp, szachownica := #szachownica) = true THEN
                   IF #poz_temp.x = #polozenie_krola.x  AND #poz_temp.y = #polozenie_krola.y  THEN
                       #sprawdz_czy_krol_szach := true;
                   END_IF;
           ELSIF "sprawdz_czy_zajete"(pozycja := #poz_temp, szachownica := #szachownica) = 2 THEN
                   IF #poz_temp.x = #polozenie_krola.x  AND #poz_temp.y = #polozenie_krola.y  THEN
                       #sprawdz_czy_krol_szach := true;
                   END_IF;
           END_IF;
       END_IF;
       #poz_temp.x := #krol.pozycja.x - 1;
       #poz_temp.y := #krol.pozycja.y;
       IF "sprawdz_czy_na_szachownicy"(#poz_temp) = true THEN
           IF "sprawdz_czy_wolne"(pozycja := #poz_temp, szachownica := #szachownica) = true THEN
                   IF #poz_temp.x = #polozenie_krola.x  AND #poz_temp.y = #polozenie_krola.y  THEN
                       #sprawdz_czy_krol_szach := true;
                   END_IF;
           ELSIF "sprawdz_czy_zajete"(pozycja := #poz_temp, szachownica := #szachownica) = 2 THEN
                   IF #poz_temp.x = #polozenie_krola.x  AND #poz_temp.y = #polozenie_krola.y  THEN
                       #sprawdz_czy_krol_szach := true;
                   END_IF;
           END_IF;
       END_IF;
       #poz_temp.x := #krol.pozycja.x - 1;
       #poz_temp.y := #krol.pozycja.y + 1;
       IF "sprawdz_czy_na_szachownicy"(#poz_temp) = true THEN
           IF "sprawdz_czy_wolne"(pozycja := #poz_temp, szachownica := #szachownica) = true THEN
                   IF #poz_temp.x = #polozenie_krola.x  AND #poz_temp.y = #polozenie_krola.y  THEN
                       #sprawdz_czy_krol_szach := true;
                   END_IF;
           ELSIF "sprawdz_czy_zajete"(pozycja := #poz_temp, szachownica := #szachownica) = 2 THEN
                   IF #poz_temp.x = #polozenie_krola.x  AND #poz_temp.y = #polozenie_krola.y  THEN
                       #sprawdz_czy_krol_szach := true;
                   END_IF;
           END_IF;
       END_IF;
   END_IF;
END_FUNCTION

FUNCTION "sprawdz_czy_hetman_szach" : Bool   // FC23, SCL
{ S7_Optimized_Access := 'TRUE' }
VERSION : 0.1
   VAR_INPUT
      szachownica : "Szachownica";
      polozenie_krola : "Pozycja";
   END_VAR
   VAR_IN_OUT
      hetman : "Figura";
   END_VAR
   VAR_TEMP
      poz_temp : "Pozycja";
      wykonuj_petle : Bool;
      indeks_mozliwych_ruchow : Int;
   END_VAR
BEGIN
   #indeks_mozliwych_ruchow := 0;
   #sprawdz_czy_hetman_szach := false;

   IF #hetman.kolor = 1 THEN
       // ruch białych 
       // 
       //ruch po skosie 
       #wykonuj_petle := TRUE;
       #poz_temp := #hetman.pozycja;
       WHILE #wykonuj_petle DO
           #poz_temp.x += 1;
           #poz_temp.y += 1;
           IF "sprawdz_czy_na_szachownicy"(#poz_temp) = true THEN
               IF "sprawdz_czy_wolne"(pozycja := #poz_temp, szachownica := #szachownica) = true THEN
                   IF #poz_temp.x = #polozenie_krola.x  AND #poz_temp.y = #polozenie_krola.y  THEN
                       #sprawdz_czy_hetman_szach := true;
                   END_IF;
               ELSIF "sprawdz_czy_zajete"(pozycja := #poz_temp, szachownica := #szachownica) = 1 THEN
                   IF #poz_temp.x = #polozenie_krola.x  AND #poz_temp.y = #polozenie_krola.y  THEN
                       #sprawdz_czy_hetman_szach := true;
                   ELSE
                       #wykonuj_petle := false;
                   END_IF;
               ELSE
                   #wykonuj_petle := false;
                END_IF;
           ELSE
               #wykonuj_petle := false;
           END_IF;
       END_WHILE;
       #wykonuj_petle := TRUE;
       #poz_temp := #hetman.pozycja;
       WHILE #wykonuj_petle DO
           #poz_temp.x += 1;
           #poz_temp.y -= 1;
           IF "sprawdz_czy_na_szachownicy"(#poz_temp) = true THEN
               IF "sprawdz_czy_wolne"(pozycja := #poz_temp, szachownica := #szachownica) = true THEN
                   IF #poz_temp.x = #polozenie_krola.x  AND #poz_temp.y = #polozenie_krola.y  THEN
                       #sprawdz_czy_hetman_szach := true;
                   END_IF;
               ELSIF "sprawdz_czy_zajete"(pozycja := #poz_temp, szachownica := #szachownica) = 1 THEN
                   IF #poz_temp.x = #polozenie_krola.x  AND #poz_temp.y = #polozenie_krola.y  THEN
                       #sprawdz_czy_hetman_szach := true;
                   ELSE
                       #wykonuj_petle := false;
                   END_IF;
               ELSE
                   #wykonuj_petle := false;
               END_IF;
           ELSE
               #wykonuj_petle := false;
           END_IF;
       END_WHILE;
       #wykonuj_petle := TRUE;
       #poz_temp := #hetman.pozycja;
       WHILE #wykonuj_petle DO
           #poz_temp.x -= 1;
           #poz_temp.y += 1;
           IF "sprawdz_czy_na_szachownicy"(#poz_temp) = true THEN
               IF "sprawdz_czy_wolne"(pozycja := #poz_temp, szachownica := #szachownica) = true THEN
                   IF #poz_temp.x = #polozenie_krola.x  AND #poz_temp.y = #polozenie_krola.y  THEN
                       #sprawdz_czy_hetman_szach := true;
                   END_IF;
               ELSIF "sprawdz_czy_zajete"(pozycja := #poz_temp, szachownica := #szachownica) = 1 THEN
                   IF #poz_temp.x = #polozenie_krola.x  AND #poz_temp.y = #polozenie_krola.y  THEN
                       #sprawdz_czy_hetman_szach := true;
                   ELSE
                       #wykonuj_petle := false;
                   END_IF;
               ELSE
                   #wykonuj_petle := false;
               END_IF;
           ELSE
               #wykonuj_petle := false;
           END_IF;
       END_WHILE;
       #wykonuj_petle := TRUE;
       #poz_temp := #hetman.pozycja;
       WHILE #wykonuj_petle DO
           #poz_temp.x -= 1;
           #poz_temp.y -= 1;
           IF "sprawdz_czy_na_szachownicy"(#poz_temp) = true THEN
               IF "sprawdz_czy_wolne"(pozycja := #poz_temp, szachownica := #szachownica) = true THEN
                   IF #poz_temp.x = #polozenie_krola.x  AND #poz_temp.y = #polozenie_krola.y  THEN
                       #sprawdz_czy_hetman_szach := true;
                   END_IF;
               ELSIF "sprawdz_czy_zajete"(pozycja := #poz_temp, szachownica := #szachownica) = 1 THEN
                   IF #poz_temp.x = #polozenie_krola.x  AND #poz_temp.y = #polozenie_krola.y  THEN
                       #sprawdz_czy_hetman_szach := true;
                   ELSE
                       #wykonuj_petle := false;
                   END_IF;
               ELSE
                   #wykonuj_petle := false;
               END_IF;
           ELSE
               #wykonuj_petle := false;
           END_IF;
       END_WHILE;
       //ruch poziomo i pionowo
       #wykonuj_petle := TRUE;
       #poz_temp := #hetman.pozycja;
       WHILE #wykonuj_petle DO
           #poz_temp.x += 1;
           #poz_temp.y += 0;
           IF "sprawdz_czy_na_szachownicy"(#poz_temp) = true THEN
               IF "sprawdz_czy_wolne"(pozycja := #poz_temp, szachownica := #szachownica) = true THEN
                   IF #poz_temp.x = #polozenie_krola.x  AND #poz_temp.y = #polozenie_krola.y  THEN
                       #sprawdz_czy_hetman_szach := true;
                   END_IF;
               ELSIF "sprawdz_czy_zajete"(pozycja := #poz_temp, szachownica := #szachownica) = 1 THEN
                   IF #poz_temp.x = #polozenie_krola.x  AND #poz_temp.y = #polozenie_krola.y  THEN
                       #sprawdz_czy_hetman_szach := true;
                   ELSE
                       #wykonuj_petle := false;
                   END_IF;
               ELSE
                   #wykonuj_petle := false;
               END_IF;
           ELSE
               #wykonuj_petle := false;
           END_IF;
       END_WHILE;
       #wykonuj_petle := TRUE;
       #poz_temp := #hetman.pozycja;
       WHILE #wykonuj_petle DO
           #poz_temp.x += 0;
           #poz_temp.y += 1;
           IF "sprawdz_czy_na_szachownicy"(#poz_temp) = true THEN
               IF "sprawdz_czy_wolne"(pozycja := #poz_temp, szachownica := #szachownica) = true THEN
                   IF #poz_temp.x = #polozenie_krola.x  AND #poz_temp.y = #polozenie_krola.y  THEN
                       #sprawdz_czy_hetman_szach := true;
                   END_IF;
               ELSIF "sprawdz_czy_zajete"(pozycja := #poz_temp, szachownica := #szachownica) = 1 THEN
                   IF #poz_temp.x = #polozenie_krola.x  AND #poz_temp.y = #polozenie_krola.y  THEN
                       #sprawdz_czy_hetman_szach := true;
                   ELSE
                       #wykonuj_petle := false;
                   END_IF;
               ELSE
                   #wykonuj_petle := false;
               END_IF;
           ELSE
               #wykonuj_petle := false;
           END_IF;
       END_WHILE;
       #wykonuj_petle := TRUE;
       #poz_temp := #hetman.pozycja;
       WHILE #wykonuj_petle DO
           #poz_temp.x += -1;
           #poz_temp.y += 0;
           IF "sprawdz_czy_na_szachownicy"(#poz_temp) = true THEN
               IF "sprawdz_czy_wolne"(pozycja := #poz_temp, szachownica := #szachownica) = true THEN
                   IF #poz_temp.x = #polozenie_krola.x  AND #poz_temp.y = #polozenie_krola.y  THEN
                       #sprawdz_czy_hetman_szach := true;
                   END_IF;
               ELSIF "sprawdz_czy_zajete"(pozycja := #poz_temp, szachownica := #szachownica) = 1 THEN
                   IF #poz_temp.x = #polozenie_krola.x  AND #poz_temp.y = #polozenie_krola.y  THEN
                       #sprawdz_czy_hetman_szach := true;
                   ELSE
                       #wykonuj_petle := false;
                   END_IF;
               ELSE
                   #wykonuj_petle := false;
               END_IF;
           ELSE
               #wykonuj_petle := false;
           END_IF;
       END_WHILE;
       #wykonuj_petle := TRUE;
       #poz_temp := #hetman.pozycja;
       WHILE #wykonuj_petle DO
           #poz_temp.x += 0;
           #poz_temp.y += -1;
           IF "sprawdz_czy_na_szachownicy"(#poz_temp) = true THEN
               IF "sprawdz_czy_wolne"(pozycja := #poz_temp, szachownica := #szachownica) = true THEN
                   IF #poz_temp.x = #polozenie_krola.x  AND #poz_temp.y = #polozenie_krola.y  THEN
                       #sprawdz_czy_hetman_szach := true;
                   END_IF;
               ELSIF "sprawdz_czy_zajete"(pozycja := #poz_temp, szachownica := #szachownica) = 1 THEN
                   IF #poz_temp.x = #polozenie_krola.x  AND #poz_temp.y = #polozenie_krola.y  THEN
                       #sprawdz_czy_hetman_szach := true;
                   ELSE
                       #wykonuj_petle := false;
                   END_IF;
               ELSE
                   #wykonuj_petle := false;
               END_IF;
           ELSE
               #wykonuj_petle := false;
           END_IF;
       END_WHILE;


